// TIA Portal V17 program export: 0 tag tables, 0 data types, 15 data blocks, 22 code blocks (in call order from the OBs), 17 instance data blocks

DATA_BLOCK "GLOBAL_DB"   // DB14
{ S7_Optimized_Access := 'TRUE' }
VERSION : 0.1
// stored: AutoNumber true, DBAccessibleFromOPCUA true, DBAccessibleFromWebserver true, IsOnlyStoredInLoadMemory false, IsRetainMemResEnabled false, IsWriteProtectedInAS false, MemoryReserve 100
   VAR
      CurrentTime : Date_And_Time;
      RS232_SendBuff : DWord;
      RS232_RecvBuff : DWord;
   END_VAR
BEGIN
END_DATA_BLOCK

DATA_BLOCK "GDB_Database"   // DB7
{ S7_Optimized_Access := 'TRUE' }
VERSION : 0.1
// stored: AutoNumber true, DBAccessibleFromOPCUA true, DBAccessibleFromWebserver true, IsOnlyStoredInLoadMemory false, IsRetainMemResEnabled false, IsWriteProtectedInAS false, MemoryReserve 100
   VAR
      Communication : Struct   // Communication_Status
         Error : Int;
         Active : Bool;
         Start : Bool;
         Function : Int;
         "Step" : Int;
         Done : Int;
      END_STRUCT;
      Condition : Struct
         Rob_PrgNmr : Int;
      END_STRUCT;
      Receive : Struct
         Rob_PRG : Int;
         Force : Real;
      END_STRUCT;
      Task_Done : Struct
         Read_from_DB : Bool;
      END_STRUCT;
      "Return" : Struct
         t : Bool;
      END_STRUCT;
      Requests : Struct
         Read_from_DB : Bool;
         Write_to_DB : Bool;
      END_STRUCT;
   END_VAR
BEGIN
END_DATA_BLOCK

DATA_BLOCK "STL_Data"   // DB2
{ S7_Optimized_Access := 'TRUE' }
VERSION : 0.1
// stored: AutoNumber true, DBAccessibleFromOPCUA true, DBAccessibleFromWebserver true, IsOnlyStoredInLoadMemory false, IsRetainMemResEnabled false, IsWriteProtectedInAS false, MemoryReserve 100
   VAR
      BasePos0 : Int;
      BasePos1 : Int;
      VarBase0 : Int;
      VarBase1 : Int;
   END_VAR
BEGIN
END_DATA_BLOCK

DATA_BLOCK "DATA_LOGGING"   // DB25
{ S7_Optimized_Access := 'TRUE' }
VERSION : 0.1
// stored: AutoNumber true, DBAccessibleFromOPCUA true, DBAccessibleFromWebserver true, IsOnlyStoredInLoadMemory false, IsRetainMemResEnabled false, IsWriteProtectedInAS false, MemoryReserve 100
   VAR
      Record : UDInt;
      "Name" : String := 'Logging';
      ID : DWord := 1;
      Header : String := 'A350-1000, Errors';
      Data : Struct
         First : UDInt;
         Second : UDInt;
         Third : UDInt;
      END_STRUCT;
   END_VAR
BEGIN
END_DATA_BLOCK

DATA_BLOCK "GDB_HMI"   // DB8
{ S7_Optimized_Access := 'TRUE' }
VERSION : 0.1
// stored: AutoNumber true, DBAccessibleFromOPCUA true, DBAccessibleFromWebserver true, IsOnlyStoredInLoadMemory false, IsRetainMemResEnabled false, IsWriteProtectedInAS false, MemoryReserve 100
   VAR
      Database : Struct
         Reset_Task : Bool;
      END_STRUCT;
      Received_Data_from_DB : Struct
         Rob_PRG : Int;
         Force : Real;
      END_STRUCT;
   END_VAR
BEGIN
END_DATA_BLOCK

DATA_BLOCK "ProjectDB78"   // DB30
{ S7_Optimized_Access := 'FALSE' }
VERSION : 0.1
// stored: AutoNumber true, DBAccessibleFromOPCUA true, DBAccessibleFromWebserver true, IsOnlyStoredInLoadMemory false, IsWriteProtectedInAS false
   VAR
      Oven_Temperature : Array[1..2100] of "OvenTemperature";
   END_VAR
BEGIN
END_DATA_BLOCK

DATA_BLOCK "ProjectDB94"   // DB29
{ S7_Optimized_Access := 'FALSE' }
VERSION : 0.1
// stored: AutoNumber true, DBAccessibleFromOPCUA true, DBAccessibleFromWebserver true, IsOnlyStoredInLoadMemory false, IsWriteProtectedInAS false
   VAR
      MainDB : "OvenTemperature";
      Req_Start { S7_SetPoint := 'True'} : Bool;
      Archive_Done : Bool;
   END_VAR
BEGIN
END_DATA_BLOCK

DATA_BLOCK "Keyence Datenausgabe"   // DB4
{ S7_Optimized_Access := 'TRUE' }
VERSION : 0.1
// stored: AutoNumber true, DBAccessibleFromOPCUA true, DBAccessibleFromWebserver true, IsOnlyStoredInLoadMemory false, IsRetainMemResEnabled false, IsWriteProtectedInAS false, MemoryReserve 100
   VAR
      Breite : Int;
      Länge : Int;
      Länge1 : Real;
      Breite1 : Real;
   END_VAR
BEGIN
END_DATA_BLOCK

DATA_BLOCK "DB_CMMT_ST"   // DB13
{ S7_Optimized_Access := 'TRUE' }
VERSION : 0.1
// stored: AutoNumber true, DBAccessibleFromOPCUA true, DBAccessibleFromWebserver true, IsOnlyStoredInLoadMemory false, IsRetainMemResEnabled false, IsWriteProtectedInAS false, MemoryReserve 100
   VAR
      "PLC -> CMMT" : "UDT_FESTO_CMMT_IN";
      "CMMT -> PLC" { S7_SetPoint := 'True'} : "UDT_FESTO_CMMT_OUT";
      ActualPos_mm { S7_SetPoint := 'True'} : Real;
      AcutalVelocity_mm_s : Real;
      SetPosition_mm : Real;
      SetVelocity_mm_s : Real := 20.0;
      HMI : Struct
         Scaled_ActualPos : Real;
         Scaled_SetpointPosition : Real;
         Scaled_ActualVelocity : Real;
      END_STRUCT;
      CLAMPING_TORQUE : Struct
         Execute : Bool;
         LinearRotative : Bool;
         ClampingTorque : Real;
         PercentForce : Real;
      END_STRUCT;
      CMMT_ST_ErrorWarningMessage : String;
   END_VAR
BEGIN
   "PLC -> CMMT".CancelTraversing := TRUE;
   "PLC -> CMMT".IntermediateStop := TRUE;
   "PLC -> CMMT".OverV := 100;
   "PLC -> CMMT".BaseSpeedValue := 0.125;
END_DATA_BLOCK

DATA_BLOCK "GDB_LJ_X8000"   // DB10
{ S7_Optimized_Access := 'TRUE' }
VERSION : 0.1
// stored: AutoNumber true, DBAccessibleFromOPCUA true, DBAccessibleFromWebserver true, IsOnlyStoredInLoadMemory false, IsRetainMemResEnabled false, IsWriteProtectedInAS false, MemoryReserve 100
   VAR
      PLC_to_LJX8000bits : "UDT_PLC --> LJ_X8000_Bits";
      PLC_to_LJX8000bytes { S7_SetPoint := 'True'} : "UDT_PLC --> LJ_X8000_Bytes";
      LJX8000_to_PLCbits { S7_SetPoint := 'True'} : "UDT_LJ_X8000 --> PLC_Bits";
      LJX8000_to_PLCbytes { S7_SetPoint := 'True'} : "UDT_LJ_X8000 --> PLC_Bytes";
      CTRL : Struct
         UserCommand : Int;
         ProgramNumber : Int;
         ResetError : Bool;
         CommandRequest : Bool;
         Trigger : Bool;
      END_STRUCT;
      HMI : Struct
         StartMeasurement : Bool;
         MeasurementMode : Bool;
         HandMode : Bool;
         CellType : SInt;
         SQ_ActivTask : SInt;
      END_STRUCT;
      Cell_MeasData : Struct
         Länge : Real;
         Breite : Real;
      END_STRUCT;
   END_VAR
BEGIN
END_DATA_BLOCK

DATA_BLOCK "Global_Data"   // DB3
{ S7_Optimized_Access := 'TRUE' }
VERSION : 0.1
// stored: AutoNumber true, DBAccessibleFromOPCUA true, DBAccessibleFromWebserver true, IsOnlyStoredInLoadMemory false, IsRetainMemResEnabled false, IsWriteProtectedInAS false, MemoryReserve 100
   VAR
      "LK-G5001P" : Struct   // Distanzsensoren - KEYENCE
         "LK-H057-01" : Real;
         "LK-H057-02" : Real;
      END_STRUCT;
      testbit : Bool;
   END_VAR
BEGIN
END_DATA_BLOCK

DATA_BLOCK "LK_G5000_DATA"   // DB16
{ S7_Optimized_Access := 'TRUE' }
VERSION : 0.1
// stored: AutoNumber true, DBAccessibleFromOPCUA true, DBAccessibleFromWebserver true, IsOnlyStoredInLoadMemory false, IsRetainMemResEnabled false, IsWriteProtectedInAS false, MemoryReserve 100
   VAR
      RS232_CTRL : Struct
         TO_LKG5000 : "UDT_LKG5000_RS232_SEND";
         FROM_LKG5000 { S7_SetPoint := 'True'} : "UDT_LKG5000_RS232_RCV";
      END_STRUCT;
      SEND_BUFF : "UDT_RS232_SEND_DATA";
      RCV_BUFF { S7_SetPoint := 'True'} : "UDT_RS232_RCV_DATA";
      RS232_Command { S7_SetPoint := 'True'} : String[11];
   END_VAR
BEGIN
END_DATA_BLOCK

DATA_BLOCK "DB_Receipe"   // DB6
{ S7_Optimized_Access := 'TRUE' }
VERSION : 0.1
// stored: AutoNumber true, DBAccessibleFromOPCUA true, DBAccessibleFromWebserver true, IsOnlyStoredInLoadMemory false, IsRetainMemResEnabled false, IsWriteProtectedInAS false, MemoryReserve 100
   VAR
      "Time" : Time;
      Temperature : Int;
      Fan : Bool;
   END_VAR
BEGIN
END_DATA_BLOCK

DATA_BLOCK "DB_ScanData"   // DB5
{ S7_Optimized_Access := 'TRUE' }
VERSION : 0.1
// stored: AutoNumber true, DBAccessibleFromOPCUA true, DBAccessibleFromWebserver true, IsOnlyStoredInLoadMemory false, IsRetainMemResEnabled false, IsWriteProtectedInAS false, MemoryReserve 100
   VAR
      ST01_MessGewichtMasse : Struct
         Request_for_Scan : Bool;
         DatenVorhanden : Bool;
         "Tray+Zelle" : Array[1..1, 1..1] of "UDT_ProGloveScanDat";
      END_STRUCT;
      ST02_EOLMessungImpdanz : Struct
         Request_for_Scan : Bool;
         DatenVoranden : Bool;
         "Tray+Zelle" : Array[1..2, 1..6] of "UDT_ProGloveScanDat";
      END_STRUCT;
      ST03_Dichtigkeitspruefung : Struct
         Request_for_Scan : Bool;
         DatenVoranden : Bool;
         "Tray+Zelle" : Array[1..1, 1..1] of "UDT_ProGloveScanDat";
      END_STRUCT;
      ST04_Degassing : Struct
         Request_for_Scan : Bool;
         DatenVorhanden : Bool;
         "Tray+Zelle" : Array[1..1, 1..1] of "UDT_ProGloveScanDat";
      END_STRUCT;
      ST05_Formierung : Struct
         Request_for_Scan : Bool;
         DatenVorhanden : Bool;
         Schrank : Array[1..2] of "UDT_Formierung";
      END_STRUCT;
      ST06_Soaking : Struct
         Request_for_Scan : Bool;
         DatenVorhanden : Bool;
         Schrank : Array[1..4] of "UDT_Formierung";
      END_STRUCT;
      ST07_Aging : Struct
         Request_for_Scan : Bool;
         DatenVorhanden : Bool;
         Schrank : Array[1..30] of "UDT_Aging";
      END_STRUCT;
      ST08_MobileOCVMessung : Struct
         Request_for_Scan : Bool;
         DatenVorhanden : Bool;
         "Tray+Zelle" : Array[1..1, 1..6] of "UDT_ProGloveScanDat";
      END_STRUCT;
   END_VAR
BEGIN
END_DATA_BLOCK

DATA_BLOCK "PROGLOVE_TCP"   // DB32
{ S7_Optimized_Access := 'TRUE' }
VERSION : 0.1
// stored: AutoNumber true, DBAccessibleFromOPCUA true, DBAccessibleFromWebserver true, IsOnlyStoredInLoadMemory false, IsRetainMemResEnabled false, IsWriteProtectedInAS false, MemoryReserve 100
   VAR
      SEND_DATA { S7_SetPoint := 'True'} : String;
      RCV_DATA : String;
      TCON : Struct
         Done : Bool;
         Busy : Bool;
         Error : Bool;
         Status : Word;
      END_STRUCT;
   END_VAR
BEGIN
END_DATA_BLOCK

ORGANIZATION_BLOCK "Main"   // OB1, LAD, ProgramCycle
TITLE = "Main Program Sweep (Cycle)"
{ S7_Optimized_Access := 'TRUE' }
VERSION : 0.1
// stored: AutoNumber true, IsIECCheckEnabled false, SetENOAutomatically false
   VAR_INPUT
      Initial_Call : Bool;   // Initial call of this OB
      Remanence : Bool;   // =True, if remanent data are available
   END_VAR
   VAR_TEMP
      RetVAl : Int;
   END_VAR
BEGIN

REGION Network 1: Read Local Time
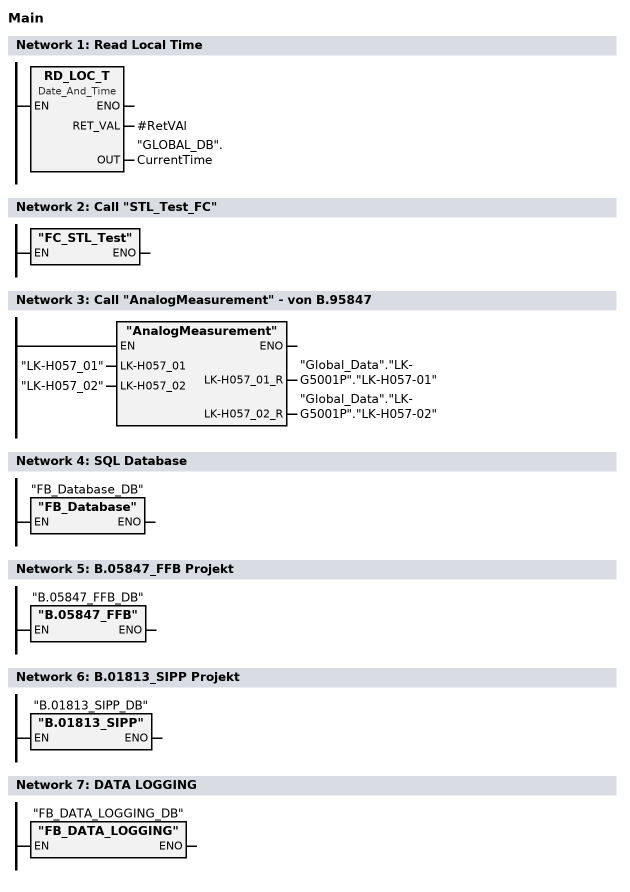
   RUNG wire#powerrail
      { S7_Templates := "date_type := Date_And_Time" } RD_LOC_T(RET_VAL => #RetVAl, OUT => "GLOBAL_DB".CurrentTime)
   END_RUNG
   // the same network as SCL:
   #RetVAl := RD_LOC_T(OUT => "GLOBAL_DB".CurrentTime);
END_REGION

REGION Network 2: Call "STL_Test_FC"
   RUNG wire#powerrail
      "FC_STL_Test"()
   END_RUNG
   // the same network as SCL:
   "FC_STL_Test"();
END_REGION

REGION Network 3: Call "AnalogMeasurement" - von B.95847
   RUNG wire#powerrail
      "AnalogMeasurement"("LK-H057_01" := "LK-H057_01", "LK-H057_02" := "LK-H057_02", "LK-H057_01_R" => "Global_Data"."LK-G5001P"."LK-H057-01", "LK-H057_02_R" => "Global_Data"."LK-G5001P"."LK-H057-02")
   END_RUNG
   // the same network as SCL:
   "AnalogMeasurement"("LK-H057_01" := "LK-H057_01",
                       "LK-H057_02" := "LK-H057_02",
                       "LK-H057_01_R" => "Global_Data"."LK-G5001P"."LK-H057-01",
                       "LK-H057_02_R" => "Global_Data"."LK-G5001P"."LK-H057-02");
END_REGION

REGION Network 4: SQL Database
   RUNG wire#powerrail
      "FB_Database_DB"()
   END_RUNG
   // the same network as SCL:
   "FB_Database_DB"();   // "FB_Database"
END_REGION

REGION Network 5: B.05847_FFB Projekt
   RUNG wire#powerrail
      "B.05847_FFB_DB"()
   END_RUNG
   // the same network as SCL:
   "B.05847_FFB_DB"();   // "B.05847_FFB"
END_REGION

REGION Network 6: B.01813_SIPP Projekt
   RUNG wire#powerrail
      "B.01813_SIPP_DB"()
   END_RUNG
   // the same network as SCL:
   "B.01813_SIPP_DB"();   // "B.01813_SIPP"
END_REGION

REGION Network 7: DATA LOGGING
   RUNG wire#powerrail
      "FB_DATA_LOGGING_DB"()
   END_RUNG
   // the same network as SCL:
   "FB_DATA_LOGGING_DB"();   // "FB_DATA_LOGGING"
END_REGION
END_ORGANIZATION_BLOCK

FUNCTION "FC_STL_Test" : Void   // FC1, STL
{ S7_Optimized_Access := 'TRUE' }
VERSION : 0.1
// stored: AutoNumber true, UDAEnableTagReadback false
BEGIN

NETWORK
TITLE = 
// Example how to Load Set values to ACC1 ( defined variable by T )
// L is for LOAD
// T is for TRANSFER the value from bottom ( L )

      L     125;
      T     "STL_Data".BasePos0;

      L     "STL_Data".VarBase1;
      T     "STL_Data".BasePos1;


END_FUNCTION

FUNCTION "AnalogMeasurement" : Void   // FC2, LAD
{ S7_Optimized_Access := 'TRUE' }
VERSION : 0.1
// stored: AutoNumber true, IsIECCheckEnabled false, SetENOAutomatically false, UDAEnableTagReadback false
   VAR_INPUT
      "LK-H057_01" : Int;   // Keyence Dist.Senz-01
      "LK-H057_02" : Int;   // Keyence Dist.Senz-01
   END_VAR
   VAR_OUTPUT
      "LK-H057_01_R" : Real;
      "LK-H057_02_R" : Real;
   END_VAR
   VAR_TEMP
      Distanz_In_Prozent_01 : Real;
      Distanz_In_Prozent_02 : Real;
   END_VAR
BEGIN

REGION Network 1: LK-H057_01 Analog Werte
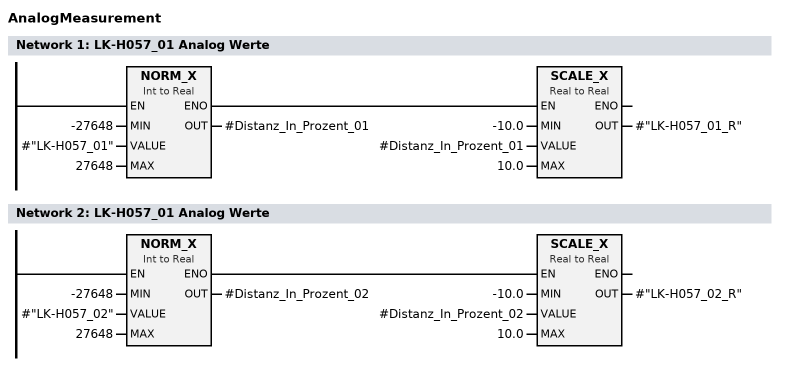
   RUNG wire#powerrail
      { S7_Templates := "[SrcType := Int, DestType := Real]" } Normalize(min := -27648, value := #"LK-H057_01", max := 27648, out => #Distanz_In_Prozent_01)
      { S7_Templates := "[SrcType := Real, DestType := Real]" } Scale(min := -10.0, value := #Distanz_In_Prozent_01, max := 10.0, out => #"LK-H057_01_R")
   END_RUNG
   // the same network as SCL:
   #Distanz_In_Prozent_01 := NORM_X(MIN := -27648, VALUE := #"LK-H057_01", MAX := 27648);
   #"LK-H057_01_R" := SCALE_X(MIN := -10.0, VALUE := #Distanz_In_Prozent_01, MAX := 10.0);
END_REGION

REGION Network 2: LK-H057_01 Analog Werte
   RUNG wire#powerrail
      { S7_Templates := "[SrcType := Int, DestType := Real]" } Normalize(min := -27648, value := #"LK-H057_02", max := 27648, out => #Distanz_In_Prozent_02)
      { S7_Templates := "[SrcType := Real, DestType := Real]" } Scale(min := -10.0, value := #Distanz_In_Prozent_02, max := 10.0, out => #"LK-H057_02_R")
   END_RUNG
   // the same network as SCL:
   #Distanz_In_Prozent_02 := NORM_X(MIN := -27648, VALUE := #"LK-H057_02", MAX := 27648);
   #"LK-H057_02_R" := SCALE_X(MIN := -10.0, VALUE := #Distanz_In_Prozent_02, MAX := 10.0);
END_REGION
END_FUNCTION

FUNCTION_BLOCK "FB_Database"   // FB2, LAD
{ S7_Optimized_Access := 'TRUE' }
VERSION : 0.1
// stored: AutoNumber true, IsIECCheckEnabled false, IsRetainMemResEnabled false, MemoryReserve 100, SetENOAutomatically false, UDAEnableTagReadback false
   VAR
      task : Int;
      Task_Start : Bool;
      TON_Act_Script { S7_SetPoint := 'True'} : TON_TIME;
   END_VAR
   VAR_TEMP
      Request : Struct
         Task_001 : Bool;
         Task_002 : Bool;
         Task_003 : Bool;
         Task_004 : Bool;
      END_STRUCT;
   END_VAR
   VAR CONSTANT
      S001_Get_Data : Int := 1;
      S002_Write_Data : Int := 2;
   END_VAR
BEGIN

NETWORK
TITLE = Reset Task Requests
// Reset Task Requests
      A     "GDB_HMI".Database.Reset_Task;
      R     "GDB_Database".Requests.Read_from_DB;
      R     "GDB_Database".Requests.Write_to_DB;



REGION Network 2 (SCL): Task Start Request
   #Request.Task_001 := "GDB_Database".Requests.Read_from_DB;
   #Request.Task_002 := "GDB_Database".Requests.Write_to_DB;
END_REGION

REGION Network 3 (SCL): 10 = Request for read Global Data
   // Set task
   IF #Request.Task_001 AND (#task = 0) THEN
       #task := 10;
   END_IF;


   //Fullfill task
   IF #task = 10 THEN

       // If reading is done
       IF "GDB_Database".Communication.Done = #S001_Get_Data AND NOT "GDB_Database".Task_Done.Read_from_DB AND "GDB_Database".Communication.Error = 0 THEN

           // Write Data from DB Receive ( on HMI Tags ) to DB on SPS
          // "GDB_HMI".Received_Data_from_DB.Rob_PRG := "GDB_Database".Receive.Rob_PRG;
          // "GDB_HMI".Received_Data_from_DB.Force := "GDB_Database".Receive.Force;
           // Set that Task is active
           "GDB_Database".Task_Done.Read_from_DB := TRUE;

       END_IF;

       // Control script
       IF #Request.Task_001 THEN
           "GDB_Database".Communication.Function := #S001_Get_Data;
           #Task_Start := TRUE;
       ELSE
           "GDB_Database".Communication.Function := 0;
           #Task_Start := FALSE;
           IF NOT "GDB_Database".Communication.Active AND "GDB_Database".Communication.Done = 0 THEN
               #task := 0;
           END_IF;
       END_IF;
   END_IF;

   // Reset Done
   IF NOT #Request.Task_001 THEN
       "GDB_Database".Task_Done.Read_from_DB := FALSE;
   END_IF;
END_REGION

REGION Network 4
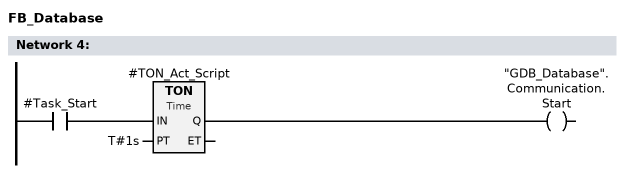
   RUNG wire#powerrail
      Contact( #Task_Start )
      { S7_Templates := "time_type := Time" } #TON_Act_Script.TON(pt := T#1s, et =>)
      Coil( "GDB_Database".Communication.Start )
   END_RUNG
   // the same network as SCL:
   #TON_Act_Script(IN := #Task_Start, PT := T#1s);   // TON
   "GDB_Database".Communication.Start := #TON_Act_Script.Q;
END_REGION
END_FUNCTION_BLOCK

FUNCTION_BLOCK "B.05847_FFB"   // FB3, LAD
{ S7_Optimized_Access := 'TRUE' }
VERSION : 0.1
// stored: AutoNumber true, IsIECCheckEnabled false, IsRetainMemResEnabled false, MemoryReserve 100, SetENOAutomatically false, UDAEnableTagReadback false
BEGIN

REGION Network 1: FESTO_CMMT_ST
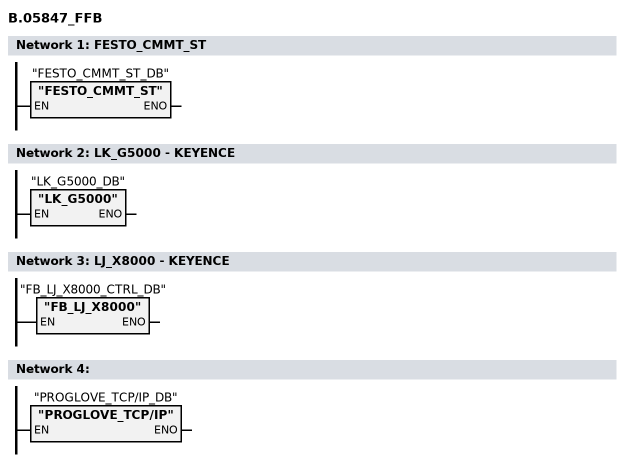
   RUNG wire#powerrail
      "FESTO_CMMT_ST_DB"()
   END_RUNG
   // the same network as SCL:
   "FESTO_CMMT_ST_DB"();   // "FESTO_CMMT_ST"
END_REGION

REGION Network 2: LK_G5000 - KEYENCE
   RUNG wire#powerrail
      "LK_G5000_DB"()
   END_RUNG
   // the same network as SCL:
   "LK_G5000_DB"();   // "LK_G5000"
END_REGION

REGION Network 3: LJ_X8000 - KEYENCE
   RUNG wire#powerrail
      "FB_LJ_X8000_CTRL_DB"()
   END_RUNG
   // the same network as SCL:
   "FB_LJ_X8000_CTRL_DB"();   // "FB_LJ_X8000"
END_REGION

REGION Network 4
   RUNG wire#powerrail
      "PROGLOVE_TCP/IP_DB"()
   END_RUNG
   // the same network as SCL:
   "PROGLOVE_TCP/IP_DB"();   // "PROGLOVE_TCP/IP"
END_REGION
END_FUNCTION_BLOCK

FUNCTION_BLOCK "FESTO_CMMT_ST"   // FB4, LAD
{ S7_Optimized_Access := 'TRUE' }
VERSION : 0.1
// stored: AutoNumber true, IsIECCheckEnabled false, IsRetainMemResEnabled false, MemoryReserve 100, SetENOAutomatically false, UDAEnableTagReadback false
   VAR
      Festo_PtP_Drives_PN_Instance { S7_SetPoint := 'True'} : "Festo_PtP_Drives_PN";
   END_VAR
   VAR_TEMP
      i : Int;
   END_VAR
BEGIN

REGION Network 1
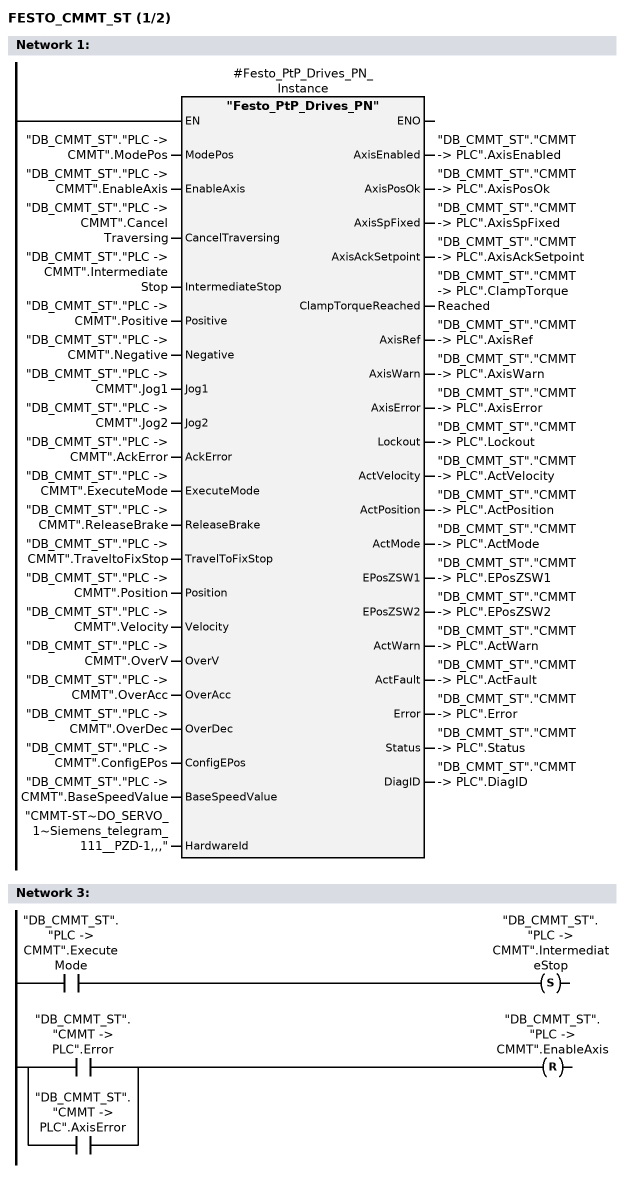
   RUNG wire#powerrail
      #Festo_PtP_Drives_PN_Instance(ModePos := "DB_CMMT_ST"."PLC -> CMMT".ModePos, EnableAxis := "DB_CMMT_ST"."PLC -> CMMT".EnableAxis, CancelTraversing := "DB_CMMT_ST"."PLC -> CMMT".CancelTraversing, IntermediateStop := "DB_CMMT_ST"."PLC -> CMMT".IntermediateStop, Positive := "DB_CMMT_ST"."PLC -> CMMT".Positive, Negative := "DB_CMMT_ST"."PLC -> CMMT".Negative, Jog1 := "DB_CMMT_ST"."PLC -> CMMT".Jog1, Jog2 := "DB_CMMT_ST"."PLC -> CMMT".Jog2, AckError := "DB_CMMT_ST"."PLC -> CMMT".AckError, ExecuteMode := "DB_CMMT_ST"."PLC -> CMMT".ExecuteMode, ReleaseBrake := "DB_CMMT_ST"."PLC -> CMMT".ReleaseBrake, TravelToFixStop := "DB_CMMT_ST"."PLC -> CMMT".TraveltoFixStop, Position := "DB_CMMT_ST"."PLC -> CMMT".Position, Velocity := "DB_CMMT_ST"."PLC -> CMMT".Velocity, OverV := "DB_CMMT_ST"."PLC -> CMMT".OverV, OverAcc := "DB_CMMT_ST"."PLC -> CMMT".OverAcc, OverDec := "DB_CMMT_ST"."PLC -> CMMT".OverDec, ConfigEPos := "DB_CMMT_ST"."PLC -> CMMT".ConfigEPos, BaseSpeedValue := "DB_CMMT_ST"."PLC -> CMMT".BaseSpeedValue, HardwareId := "CMMT-ST~DO_SERVO_1~Siemens_telegram_111__PZD-1,,,", AxisEnabled => "DB_CMMT_ST"."CMMT -> PLC".AxisEnabled, AxisPosOk => "DB_CMMT_ST"."CMMT -> PLC".AxisPosOk, AxisSpFixed => "DB_CMMT_ST"."CMMT -> PLC".AxisSpFixed, AxisAckSetpoint => "DB_CMMT_ST"."CMMT -> PLC".AxisAckSetpoint, ClampTorqueReached => "DB_CMMT_ST"."CMMT -> PLC".ClampTorqueReached, AxisRef => "DB_CMMT_ST"."CMMT -> PLC".AxisRef, AxisWarn => "DB_CMMT_ST"."CMMT -> PLC".AxisWarn, AxisError => "DB_CMMT_ST"."CMMT -> PLC".AxisError, Lockout => "DB_CMMT_ST"."CMMT -> PLC".Lockout, ActVelocity => "DB_CMMT_ST"."CMMT -> PLC".ActVelocity, ActPosition => "DB_CMMT_ST"."CMMT -> PLC".ActPosition, ActMode => "DB_CMMT_ST"."CMMT -> PLC".ActMode, EPosZSW1 => "DB_CMMT_ST"."CMMT -> PLC".EPosZSW1, EPosZSW2 => "DB_CMMT_ST"."CMMT -> PLC".EPosZSW2, ActWarn => "DB_CMMT_ST"."CMMT -> PLC".ActWarn, ActFault => "DB_CMMT_ST"."CMMT -> PLC".ActFault, Error => "DB_CMMT_ST"."CMMT -> PLC".Error, Status => "DB_CMMT_ST"."CMMT -> PLC".Status, DiagID => "DB_CMMT_ST"."CMMT -> PLC".DiagID)
   END_RUNG
   // the same network as SCL:
   #Festo_PtP_Drives_PN_Instance(ModePos := "DB_CMMT_ST"."PLC -> CMMT".ModePos,   // "Festo_PtP_Drives_PN"
                           EnableAxis := "DB_CMMT_ST"."PLC -> CMMT".EnableAxis,
                           CancelTraversing := "DB_CMMT_ST"."PLC -> CMMT".CancelTraversing,
                           IntermediateStop := "DB_CMMT_ST"."PLC -> CMMT".IntermediateStop,
                           Positive := "DB_CMMT_ST"."PLC -> CMMT".Positive,
                           Negative := "DB_CMMT_ST"."PLC -> CMMT".Negative,
                           Jog1 := "DB_CMMT_ST"."PLC -> CMMT".Jog1,
                           Jog2 := "DB_CMMT_ST"."PLC -> CMMT".Jog2,
                           AckError := "DB_CMMT_ST"."PLC -> CMMT".AckError,
                           ExecuteMode := "DB_CMMT_ST"."PLC -> CMMT".ExecuteMode,
                           ReleaseBrake := "DB_CMMT_ST"."PLC -> CMMT".ReleaseBrake,
                           TravelToFixStop := "DB_CMMT_ST"."PLC -> CMMT".TraveltoFixStop,
                           Position := "DB_CMMT_ST"."PLC -> CMMT".Position,
                           Velocity := "DB_CMMT_ST"."PLC -> CMMT".Velocity,
                           OverV := "DB_CMMT_ST"."PLC -> CMMT".OverV,
                           OverAcc := "DB_CMMT_ST"."PLC -> CMMT".OverAcc,
                           OverDec := "DB_CMMT_ST"."PLC -> CMMT".OverDec,
                           ConfigEPos := "DB_CMMT_ST"."PLC -> CMMT".ConfigEPos,
                           BaseSpeedValue := "DB_CMMT_ST"."PLC -> CMMT".BaseSpeedValue,
                           HardwareId := "CMMT-ST~DO_SERVO_1~Siemens_telegram_111__PZD-1,,,",
                           AxisEnabled => "DB_CMMT_ST"."CMMT -> PLC".AxisEnabled,
                           AxisPosOk => "DB_CMMT_ST"."CMMT -> PLC".AxisPosOk,
                           AxisSpFixed => "DB_CMMT_ST"."CMMT -> PLC".AxisSpFixed,
                           AxisAckSetpoint => "DB_CMMT_ST"."CMMT -> PLC".AxisAckSetpoint,
                           ClampTorqueReached => "DB_CMMT_ST"."CMMT -> PLC".ClampTorqueReached,
                           AxisRef => "DB_CMMT_ST"."CMMT -> PLC".AxisRef,
                           AxisWarn => "DB_CMMT_ST"."CMMT -> PLC".AxisWarn,
                           AxisError => "DB_CMMT_ST"."CMMT -> PLC".AxisError,
                           Lockout => "DB_CMMT_ST"."CMMT -> PLC".Lockout,
                           ActVelocity => "DB_CMMT_ST"."CMMT -> PLC".ActVelocity,
                           ActPosition => "DB_CMMT_ST"."CMMT -> PLC".ActPosition,
                           ActMode => "DB_CMMT_ST"."CMMT -> PLC".ActMode,
                           EPosZSW1 => "DB_CMMT_ST"."CMMT -> PLC".EPosZSW1,
                           EPosZSW2 => "DB_CMMT_ST"."CMMT -> PLC".EPosZSW2,
                           ActWarn => "DB_CMMT_ST"."CMMT -> PLC".ActWarn,
                           ActFault => "DB_CMMT_ST"."CMMT -> PLC".ActFault,
                           Error => "DB_CMMT_ST"."CMMT -> PLC".Error,
                           Status => "DB_CMMT_ST"."CMMT -> PLC".Status,
                           DiagID => "DB_CMMT_ST"."CMMT -> PLC".DiagID);
END_REGION

REGION Network 2 (SCL): Convert Veolocity and Position in mm/s and mm
   REGION Convert Setposition from mm TO 1000_Unit
       "DB_CMMT_ST"."PLC -> CMMT".Position   := REAL_TO_DINT("DB_CMMT_ST".SetPosition_mm * 1000.0);
       "DB_CMMT_ST".HMI.Scaled_SetpointPosition := "DB_CMMT_ST".SetPosition_mm / 100.0;
   END_REGION

   REGION Convert Setvelocity 
       "DB_CMMT_ST"."PLC -> CMMT".Velocity := REAL_TO_DINT("DB_CMMT_ST".SetVelocity_mm_s);
   END_REGION

   REGION Convert Actual Position from 1000Unit to mm
       "DB_CMMT_ST".ActualPos_mm := "DB_CMMT_ST"."CMMT -> PLC".ActPosition / 1000.0;
       // Scale actual position for HMI
       "DB_CMMT_ST".HMI.Scaled_ActualPos := "DB_CMMT_ST".ActualPos_mm / 100; // Value in cm
   END_REGION

   REGION Convert Actual velocity from 1000Unit TO mm/s
       "DB_CMMT_ST".AcutalVelocity_mm_s := "DB_CMMT_ST"."CMMT -> PLC".ActVelocity * 1000.0;
   END_REGION
END_REGION

REGION Network 3
   RUNG wire#powerrail
      Contact( "DB_CMMT_ST"."PLC -> CMMT".ExecuteMode )
      S_Coil( "DB_CMMT_ST"."PLC -> CMMT".IntermediateStop )
   END_RUNG
   RUNG wire#powerrail
      Contact( "DB_CMMT_ST"."CMMT -> PLC".Error )
      wire#w1
      R_Coil( "DB_CMMT_ST"."PLC -> CMMT".EnableAxis )
   END_RUNG
   RUNG wire#powerrail
      Contact( "DB_CMMT_ST"."CMMT -> PLC".AxisError )
   END_RUNG wire#w1
   // the same network as SCL:
   IF "DB_CMMT_ST"."PLC -> CMMT".ExecuteMode THEN
       "DB_CMMT_ST"."PLC -> CMMT".IntermediateStop := TRUE;
   END_IF;
   IF "DB_CMMT_ST"."CMMT -> PLC".Error OR "DB_CMMT_ST"."CMMT -> PLC".AxisError THEN
       "DB_CMMT_ST"."PLC -> CMMT".EnableAxis := FALSE;
   END_IF;
END_REGION

REGION Network 4: Festo Calmping Torque
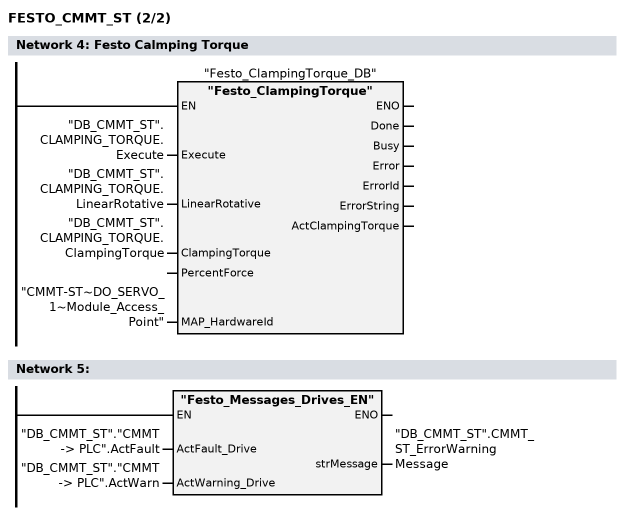
   RUNG wire#powerrail
      "Festo_ClampingTorque_DB"(Execute := "DB_CMMT_ST".CLAMPING_TORQUE.Execute, LinearRotative := "DB_CMMT_ST".CLAMPING_TORQUE.LinearRotative, ClampingTorque := "DB_CMMT_ST".CLAMPING_TORQUE.ClampingTorque, PercentForce :=, MAP_HardwareId := "CMMT-ST~DO_SERVO_1~Module_Access_Point", Done =>, Busy =>, Error =>, ErrorId =>, ErrorString =>, ActClampingTorque =>)
   END_RUNG
   // the same network as SCL:
   "Festo_ClampingTorque_DB"(Execute := "DB_CMMT_ST".CLAMPING_TORQUE.Execute,   // "Festo_ClampingTorque"
                           LinearRotative := "DB_CMMT_ST".CLAMPING_TORQUE.LinearRotative,
                           ClampingTorque := "DB_CMMT_ST".CLAMPING_TORQUE.ClampingTorque,
                           MAP_HardwareId := "CMMT-ST~DO_SERVO_1~Module_Access_Point");
END_REGION

REGION Network 5
   RUNG wire#powerrail
      "Festo_Messages_Drives_EN"(ActFault_Drive := "DB_CMMT_ST"."CMMT -> PLC".ActFault, ActWarning_Drive := "DB_CMMT_ST"."CMMT -> PLC".ActWarn, strMessage => "DB_CMMT_ST".CMMT_ST_ErrorWarningMessage)
   END_RUNG
   // the same network as SCL:
   "Festo_Messages_Drives_EN"(ActFault_Drive := "DB_CMMT_ST"."CMMT -> PLC".ActFault,
                           ActWarning_Drive := "DB_CMMT_ST"."CMMT -> PLC".ActWarn,
                           strMessage => "DB_CMMT_ST".CMMT_ST_ErrorWarningMessage);
END_REGION
END_FUNCTION_BLOCK

FUNCTION_BLOCK "Festo_PtP_Drives_PN"
TITLE = PtP function block for positioning with Tel111
{ S7_Optimized_Access := 'TRUE' }
AUTHOR : Festo
FAMILY : 'E-.Drives'
VERSION : 1.5
   VAR_INPUT 
      ModePos : Int := 0;   //   Settings of the mode
      EnableAxis : Bool := 0;   //   1 = Enable the drive
      CancelTraversing : Bool := 1;   //   0 = Reject active traverse task
      IntermediateStop : Bool := 1;   //   0 = IntermediateStop
      Positive : Bool := 0;   //   1 = Modulo positive
      Negative : Bool := 0;   //   1 = Modulo negative
      Jog1 : Bool := 0;   //   1 = jog positive
      Jog2 : Bool := 0;   //   1 = jog negative
      AckError : Bool := 0;   //   1  = Acknowledge of errors
      ExecuteMode : Bool := 0;   //   0-->1 = Start the mode
      ReleaseBrake : Bool := 0;   //   1 = Release Brake 0 = close
      TravelToFixStop : Bool := 0;   //   1 = Activation TravelToFixStop
      Position : DInt := 0;   //   Position of the MDI mode or setting of traversing block
      Velocity : DInt := 0;   //   MDI velocity
      OverV : Int := 100;   //   Override of  velocity in [%] --> 4000h=100%
      OverAcc : Int := 100;   //   Override of acceleration in [%] --> 4000h=100%
      OverDec : Int := 100;   //   Override of deceleration in [%] --> 4000h=100%
      ConfigEPos : DWord := 16#0000_000F;   //   binary programmed input -> see manual
      BaseSpeedValue : Real;   //   Value for scaling the RPM display value
      HardwareId : HW_IO := 0;   //   Hardware Identifer
   END_VAR

   VAR_OUTPUT 
      AxisEnabled : Bool := 0;   //   1= Axis in operation
      AxisPosOk : Bool := 0;   //   1= Position setpoint reached
      AxisSpFixed : Bool := 0;   //   1= Drive at standstill
      AxisAckSetpoint : Bool := 0;   //   1= Acknowledge setpoint
      ClampTorqueReached : Bool;   //   1= Clamping torque is reached
      AxisRef : Bool := 0;   //   1= Reference point set
      AxisWarn : Bool := 0;   //   1= Axis warning present
      AxisError : Bool := 0;   //   1= Axis fault present
      Lockout : Bool := 0;   //   1= Axis in lockout state
      ActVelocity : Real := 0.0;   //   Actual drive speed (has to be normed with PNU60000 --> 40000000h = 100%, if BaseSpeedValue is <> 0)
      ActPosition : DInt := 0;   //   Actual position in user unit
      ActMode : Int := 0;   //   Active ModePos mode
      EPosZSW1 : Word := 0;   //   Status of EPOS ZSW1
      EPosZSW2 : Word := 0;   //   Status of EPOS ZSW2
      ActWarn : Word := 0;   //   Actual number of warning
      ActFault : Word := 0;   //   Actual number of error
      Error : Bool := 0;   //   1 = Error present
      Status : Word := 0;   //   Status output (7002 = FB in operation; 8xxx = error description  - read the manual)
      DiagID : Word := 0;   //   Error codes of the cyclic system funtion blocks DPWR / DPRD_DAT
   END_VAR

   VAR 
      stat_Ready4Motion : Bool := 0;   // 1= drive is ready for a new set command
      stat_ExecuteIntern : Bool := 0;   // Internal ExecuteMode signal
      stat_StepHome : UInt;   // step variable for homing
      stat_RetDPRD : Int;   // Static return value for DPRD_DAT
      stat_RetDPWR : Int;   // Static return value for DPWR_DAT
      stat_CycWrite : Struct   // Structure representing the send direction (PLC to drive)
         STW1 : Struct
            jog1 : Bool;   // Bit8
            jog2 : Bool;   // Bit9
            controlByPlc : Bool := TRUE;   // Bit10
            StartHoming : Bool;   // Bit11
            ReleaseBrake : Bool;   // Bit12
            ExternalBlockChange : Bool;   // Bit13
            reserved14 : Bool;   // Bit14
            reserved15 : Bool;   // Bit15
            on : Bool;   // Bit0
            noCoastStop : Bool := TRUE;   // Bit1
            noQuickStop : Bool := TRUE;   // Bit2
            enableOperation : Bool := TRUE;   // Bit3
            cancelTraversing : Bool;   // Bit4
            intermediateStop : Bool;   // Bit5
            activateTraversing : Bool;   // Bit6
            acknowledgeFault : Bool;   // Bit7
         END_STRUCT;
         POS_STW1 : Struct
            MDI_MOD : Bool;   // Bit 8, 1= absolut, 0=relative
            PosModulo : Bool;   // Bit 9, 1=positive direction
            NegModulo : Bool;   // Bit 10, 1=negative direction
            reserved11 : Bool;   // Bit 11
            reserved12 : Bool;   // Bit 12
            reserved13 : Bool;   // Bit 13
            SetupMode : Bool;   // Bit 14, 1=Setup mode activation
            MDI_Activate : Bool;   // Bit 15, 1 =MDI mode activation
            travBlockBit0 : Bool;   // Bit 0
            travBlockBit1 : Bool;   // Bit 1
            travBlockBit2 : Bool;   // Bit 2
            travBlockBit3 : Bool;   // Bit 3
            travBlockBit4 : Bool;   // Bit 4
            travBlockBit5 : Bool;   // Bit 5
            travBlockBit6 : Bool;   // Bit 6
            reserved7 : Bool;   // Bit 7
         END_STRUCT;
         POS_STW2 : Struct
            FlyingRef : Bool;   // Bit 8, 1=Flying referencing activation
            reserved9 : Bool;   // Bit 9,
            SelectProbe : Bool;   // Bit 10, 0=Probe1, 1=Probe2
            ProbeEdgeEval : Bool;   // Bit 11, 0=rising edge, 1=falling edge
            reserved12 : Bool;   // Bit 12
            reserved13 : Bool;   // Bit 13
            "SW-Limit" : Bool;   // Bit 14, 1=Activation of SW-limits
            "HW-Limit" : Bool;   // Bit 15, 1 =Activation of HW-limits
            Trackingmode : Bool;   // Bit 0, 1=Trackingmode
            SetReferencePoint : Bool;   // Bit 1, 1=set reference point
            reserved2 : Bool;   // Bit 2
            reserved3 : Bool;   // Bit 3
            reserved4 : Bool;   // Bit 4
            jog_inc : Bool;   // Bit 5, 1=jog incremental
            reserved6 : Bool;   // Bit 6
            reserved7 : Bool;   // Bit 7
         END_STRUCT;
         STW2 : Struct
            TravelToFixStop : Bool;   // Bit8
            reserved9 : Bool;
            reserved10 : Bool;
            reserved11 : Bool;
            signOfLifeBit0 : Bool;   // Bit12
            signOfLifeBit1 : Bool;   // Bit 13
            signOfLifeBit2 : Bool;   // Bit 14
            signOfLifeBit3 : Bool;   // Bit 15
            reserved0 : Bool;
            reserved1 : Bool;
            reserved2 : Bool;
            reserved3 : Bool;
            reserved4 : Bool;
            reserved5 : Bool;
            reserved6 : Bool;
            reserved7 : Bool;
         END_STRUCT;
         Override : Word;
         MDI_TARPOS : DInt;
         MDI_VELOCITY : DInt;
         MDI_ACC : UInt;
         MDI_DEC : UInt;
         reserved11 : Word;
      END_STRUCT;
      stat_CycRead : Struct   // Structure representing the receiving direction (PLC from drive)
         ZSW1 : Struct
            followingErrorInTolerance : Bool;   // Bit 8
            controlRequest : Bool;   // Bit 9
            targetPosReached : Bool;   // Bit10
            homePosSet : Bool;   // Bit 11
            acknowledgeTraversingBlockActivated : Bool;   // Bit 12
            driveStopped : Bool;   // Bit 13
            axisAccelerates : Bool;   // Bit 14
            axisDecelerates : Bool;   // Bit 15
            readyForSwitchOn : Bool;   // Bit 0
            ready : Bool;   // Bit 1
            operationEnabled : Bool;   // Bit 2
            faultPresent : Bool;   // Bit 3
            noCoastingActive : Bool;   // Bit 4
            noQuickStopActive : Bool;   // Bit 5
            switchingOnInhibitedActive : Bool;   // Bit 6
            warningActive : Bool;   // Bit 7
         END_STRUCT;
         POS_ZSW1 : Word;
         POS_ZSW2 : Word;
         ZSW2 : Struct
            deviceSpecificBit8 : Bool;
            deviceSpecificBit9 : Bool;
            deviceSpecificBit10 : Bool;
            deviceSpecificBit11 : Bool;
            doSignOfLifeBit0 : Bool;
            doSignOfLifeBit1 : Bool;
            doSignOfLifeBit2 : Bool;
            doSignOfLifeBit3 : Bool;
            deviceSpecificBit0 : Bool;
            deviceSpecificBit1 : Bool;
            deviceSpecificBit2 : Bool;
            deviceSpecificBit3 : Bool;
            deviceSpecificBit4 : Bool;
            deviceSpecificBit5 : Bool;
            deviceSpecificBit6 : Bool;
            deviceSpecificBit7 : Bool;
         END_STRUCT;
         MELDW : Word;
         XIST_A : DInt;
         NIST_B : DInt;
         Fault_Code : Word;
         Warn_Code : Word;
         Reserved : Word;
      END_STRUCT;
      stat_ExecAux : Bool;
      stat_ExecR_Trig : Bool;
      stat_Jog1PAux : Bool;
      stat_Jog1PR_trig : Bool;
      stat_Jog2PAux : Bool;
      stat_Jog2PR_trig : Bool;
      stat_Jog1PMode8Aux : Bool;
      stat_Jog1PMode8R_trig : Bool;
      stat_Jog2PMode8Aux : Bool;
      stat_Jog2PMode8R_trig : Bool;
      stat_Status : Word;
      statStartCounter : Int;
      stat_ActMode : Int;
      stat_MaxCounterRetries { ExternalAccessible := 'False'; ExternalVisible := 'False'; ExternalWritable := 'False'} : Int;   // Maximum amount of retries for StartTask
   END_VAR

   VAR_TEMP 
      tempDWord : DWord;   // DWORD for calculation
      tmpSendBuffer : Array[0..11] of Word;   // Buffer to write
      tmpReadBuffer : Array[0..11] of Word;   // Buffer to read
   END_VAR

   VAR CONSTANT 
      MaxCounterStart : Int := 50;   // Maximum cycles for checking ACKStart
      MAXMODE : Int := 8;   // Maximum allowable mode
      STATUS_IN_OPERATION : Word := 16#7002;   // Function block Operational
      ERROR_INVALID_MODE : Word := 16#8202;   // Invalid Mode of Operation selected
      ERROR_OVERRIDE : Word := 16#8203;   // Invalid Override Value
      ERROR_INVALID_TRV_BLOCK : Word := 16#8204;   // Invalid traversing block
      ERROR_DRIVE_ERROR : Word := 16#8401;   // Drive fault
      ERROR_SWITCH_ON_INHIBITED : Word := 16#8402;   // Switch on inhibited
      ERROR_DPRD_DAT : Word := 16#8600;   // Error reading telegram data
      ERROR_DPWR_DAT : Word := 16#8601;   // Error writing telegram data
   END_VAR


BEGIN
	(*############################################################
	    FESTO SE & Co. KG, Esslingen
	    Copyright (c) 2020. All rights reserved.    
	
	    NAME OF FUNCTION BLOCK:         Festo_PTP_Drives_PN
	    VERSION NUMBER:                 V1.5
	    COMPOSER:                       Festo
	    
	    -----------------------------------------------------
	   Date        Name                Activity                                                                              
	   19.03.2020  bkle                created (V1.0)
	   09.03.2021  bkle                name changed
	   18.03.2021  bkle                changed jog behaviour
	   30.07.2021  bkle                Send the StartTask again if ACK is not received - not released
	   06.08.2021  bkle                StartTask is TRUE until ExecuteMode will switch to FALSE
	   22.09.2021  bkle                Added ConfigEpos bits for ReleaseBrake and TravelToFixStop 
	############################################################*)
	
	REGION Check OPM and Override Values
	    // Check the Mode of Operation
	    IF #ModePos > #MAXMODE THEN
	        #Error := True;
	        #stat_Status := #ERROR_INVALID_MODE;
	        #stat_ExecuteIntern := false;
	    ELSIF #ModePos < 1 THEN
	        #Error := True;
	        #stat_Status := #ERROR_INVALID_MODE;
	        #stat_ExecuteIntern := false;
	    ELSE
	        IF #stat_Status = #ERROR_INVALID_MODE THEN
	            #stat_Status := #STATUS_IN_OPERATION;
	            #Error := False;
	        END_IF;
	    END_IF;
	    
	    
	    //Check the Velocity Override 
	    IF (#OverV < 0) OR (#OverV > 199) THEN
	        #stat_Status := #ERROR_OVERRIDE;
	        #Error := True;
	    ELSE
	        // Write Velocity Override into Send Buffer
	        #stat_CycWrite.Override := INT_TO_WORD(REAL_TO_INT(16384.0 * (INT_TO_REAL(#OverV) / 100.0)));
	        IF #stat_Status = #ERROR_OVERRIDE THEN
	            #stat_Status := #STATUS_IN_OPERATION;
	            #Error := False;
	        END_IF;
	    END_IF;
	    
	    //Check the Acceleration Override  (0% - 100%, 100% => W#16#4000)
	    IF (#OverAcc < 0) OR (#OverAcc > 100) THEN
	        #stat_Status := #ERROR_OVERRIDE;
	        #Error := True;
	    ELSE
	        // Write Acceleration Override into Send Buffer
	        #stat_CycWrite.MDI_ACC := INT_TO_WORD(REAL_TO_INT(16384.0 * (INT_TO_REAL(#OverAcc) / 100.0)));
	        IF #stat_Status = #ERROR_OVERRIDE THEN
	            #stat_Status := #STATUS_IN_OPERATION;
	            #Error := False;
	        END_IF;
	    END_IF;
	    
	    //Check the Deceleration Override  (0% - 100%, 100% => W#16#4000)
	    IF (#OverDec < 0) OR (#OverDec > 100) THEN
	        #stat_Status := #ERROR_OVERRIDE;
	        #Error := True;
	    ELSE
	        // Write Deceleration Override into Send Buffer
	        #stat_CycWrite.MDI_DEC := INT_TO_WORD(REAL_TO_INT(16384.0 * (INT_TO_REAL(#OverDec) / 100.0)));
	        IF #stat_Status = #ERROR_OVERRIDE THEN
	            #stat_Status := #STATUS_IN_OPERATION;
	            #Error := False;
	        END_IF;
	    END_IF;
	END_REGION ;
	
	REGION Read Cyclic Data of Telegramm111
	    // Read cyclic telegram 111
	    #stat_RetDPRD := DPRD_DAT(LADDR := #HardwareId,
	                              RECORD => #tmpReadBuffer);
	    
	    //check if the return code is unequal zero -> error occured
	    IF #stat_RetDPRD <> 0 THEN
	        #Error := true;
	        #stat_Status := #ERROR_DPRD_DAT;
	        #DiagID := INT_TO_WORD(#stat_RetDPRD);
	    ELSE
	        
	        // set the Diag status back "in operation"
	        IF #stat_Status = #ERROR_DPRD_DAT THEN
	            #stat_Status := #STATUS_IN_OPERATION;
	            #DiagID := 0;
	            #Error := False;
	        END_IF;
	    END_IF;
	    
	END_REGION ;
	
	
	REGION Read Input from temp data
	    // copy all values from tmp buffer to static data
	    // ZSW1
	    #stat_CycRead.ZSW1.followingErrorInTolerance := #tmpReadBuffer[0].%X8;
	    #stat_CycRead.ZSW1.controlRequest := #tmpReadBuffer[0].%X9;
	    #stat_CycRead.ZSW1.targetPosReached := #tmpReadBuffer[0].%X10;
	    #stat_CycRead.ZSW1.homePosSet := #tmpReadBuffer[0].%X11;
	    #stat_CycRead.ZSW1.acknowledgeTraversingBlockActivated := #tmpReadBuffer[0].%X12;
	    #stat_CycRead.ZSW1.driveStopped := #tmpReadBuffer[0].%X13;
	    #stat_CycRead.ZSW1.axisAccelerates := #tmpReadBuffer[0].%X14;
	    #stat_CycRead.ZSW1.axisDecelerates := #tmpReadBuffer[0].%X15;
	    #stat_CycRead.ZSW1.readyForSwitchOn := #tmpReadBuffer[0].%X0;
	    #stat_CycRead.ZSW1.ready := #tmpReadBuffer[0].%X1;
	    #stat_CycRead.ZSW1.operationEnabled := #tmpReadBuffer[0].%X2;
	    #stat_CycRead.ZSW1.faultPresent := #tmpReadBuffer[0].%X3;
	    #stat_CycRead.ZSW1.noCoastingActive := #tmpReadBuffer[0].%X4;
	    #stat_CycRead.ZSW1.noQuickStopActive := #tmpReadBuffer[0].%X5;
	    #stat_CycRead.ZSW1.switchingOnInhibitedActive := #tmpReadBuffer[0].%X6;
	    #stat_CycRead.ZSW1.warningActive := #tmpReadBuffer[0].%X7;
	    
	    //POS_ZSW1
	    #stat_CycRead.POS_ZSW1 := #tmpReadBuffer[1];
	    #EPosZSW1 := #stat_CycRead.POS_ZSW1;
	    
	    //POS_ZSW2
	    #stat_CycRead.POS_ZSW2 := #tmpReadBuffer[2];
	    #EPosZSW2 := #stat_CycRead.POS_ZSW2;
	    
	    // ZSW2
	    #stat_CycRead.ZSW2.deviceSpecificBit8 := #tmpReadBuffer[3].%X8;
	    #stat_CycRead.ZSW2.deviceSpecificBit9 := #tmpReadBuffer[3].%X9;
	    #stat_CycRead.ZSW2.deviceSpecificBit10 := #tmpReadBuffer[3].%X10;
	    #stat_CycRead.ZSW2.deviceSpecificBit11 := #tmpReadBuffer[3].%X11;
	    #stat_CycRead.ZSW2.doSignOfLifeBit0 := #tmpReadBuffer[3].%X12;
	    #stat_CycRead.ZSW2.doSignOfLifeBit1 := #tmpReadBuffer[3].%X13;
	    #stat_CycRead.ZSW2.doSignOfLifeBit2 := #tmpReadBuffer[3].%X14;
	    #stat_CycRead.ZSW2.doSignOfLifeBit3 := #tmpReadBuffer[3].%X15;
	    #stat_CycRead.ZSW2.deviceSpecificBit0 := #tmpReadBuffer[3].%X0;
	    #stat_CycRead.ZSW2.deviceSpecificBit1 := #tmpReadBuffer[3].%X1;
	    #stat_CycRead.ZSW2.deviceSpecificBit2 := #tmpReadBuffer[3].%X2;
	    #stat_CycRead.ZSW2.deviceSpecificBit3 := #tmpReadBuffer[3].%X3;
	    #stat_CycRead.ZSW2.deviceSpecificBit4 := #tmpReadBuffer[3].%X4;
	    #stat_CycRead.ZSW2.deviceSpecificBit5 := #tmpReadBuffer[3].%X5;
	    #stat_CycRead.ZSW2.deviceSpecificBit6 := #tmpReadBuffer[3].%X6;
	    #stat_CycRead.ZSW2.deviceSpecificBit7 := #tmpReadBuffer[3].%X7;
	    
	    //MELDW
	    #stat_CycRead.MELDW := #tmpReadBuffer[4];
	    
	    //XIST_A
	    #stat_CycRead.XIST_A.%W0 := #tmpReadBuffer[6];
	    #stat_CycRead.XIST_A.%W1 := #tmpReadBuffer[5];
	    
	    //NIST_B
	    #stat_CycRead.NIST_B.%W0 := #tmpReadBuffer[8];
	    #stat_CycRead.NIST_B.%W1 := #tmpReadBuffer[7];
	    
	    //Fault_Code
	    #stat_CycRead.Fault_Code := #tmpReadBuffer[9];
	    
	    //Warn_Code
	    #stat_CycRead.Warn_Code := #tmpReadBuffer[10];
	    
	    //Reserved
	    #stat_CycRead.Reserved := #tmpReadBuffer[11];
	END_REGION ;
	
	// Mapping of the FB Outputs
	#AxisEnabled := #stat_CycRead.ZSW1.operationEnabled;
	#AxisError := #stat_CycRead.ZSW1.faultPresent;
	#AxisWarn := #stat_CycRead.ZSW1.warningActive;
	#AxisPosOk := #stat_CycRead.ZSW1.targetPosReached;
	#AxisRef := #stat_CycRead.ZSW1.homePosSet;
	#AxisAckSetpoint := #stat_CycRead.ZSW1.acknowledgeTraversingBlockActivated;
	#ClampTorqueReached := #stat_CycRead.POS_ZSW2.%X13;
	#AxisSpFixed := #stat_CycRead.ZSW1.driveStopped;
	#ActVelocity := #stat_CycRead.NIST_B;
	
	
	//scaling the ActVelocity output
	IF #BaseSpeedValue <> 0 THEN
	    #ActVelocity := #ActVelocity * ((#BaseSpeedValue / 1073741824.0));
	END_IF;
	
	#ActPosition := #stat_CycRead.XIST_A;
	#ActWarn := #stat_CycRead.Warn_Code;
	#ActFault := #stat_CycRead.Fault_Code;
	#Lockout := #stat_CycRead.ZSW1.switchingOnInhibitedActive;
	
	//Check the drive error and Lockout status
	IF #AxisError THEN
	    #stat_Status := #ERROR_DRIVE_ERROR;
	    #Error := True;
	ELSIF #Lockout THEN
	    #stat_Status := #ERROR_SWITCH_ON_INHIBITED;
	    #Error := True;
	ELSE
	    // error is gone -> set status in operational
	    IF (#stat_Status = #ERROR_DRIVE_ERROR) OR #stat_Status = #ERROR_SWITCH_ON_INHIBITED THEN
	        #stat_Status := #STATUS_IN_OPERATION;
	        #Error := False;
	    END_IF;
	END_IF;
	
	//Enable the Axis
	#stat_CycWrite.STW1.on := #EnableAxis;                       //STW1.0
	
	//fix values for STW1 data
	#stat_CycWrite.STW1.cancelTraversing := #CancelTraversing;   //STW1.4
	#stat_CycWrite.STW1.intermediateStop := #IntermediateStop;   //STW1.5
	#stat_CycWrite.STW1.acknowledgeFault := #AckError;           //STW1.7
	#stat_CycWrite.STW1.controlByPlc := TRUE;                    //STW1.10
	#stat_CycWrite.STW1.enableOperation := TRUE;                 //STW1.3
	
	// copy the position set value into the send struct
	IF #ModePos <> 4 OR #ModePos <> 5 OR #ModePos <> 6 OR #ModePos <> 7 OR #ModePos <> 8 THEN
	    #stat_CycWrite.MDI_TARPOS := #Position;
	ELSE
	    #stat_CycWrite.MDI_TARPOS := 0;
	END_IF;
	
	//copy the velocity set value into the send struct
	#stat_CycWrite.MDI_VELOCITY := #Velocity;
	
	//Jog bits
	// Mode 7
	//Generate the Jog1 Edge
	#stat_Jog1PR_trig := #Jog1 AND NOT #stat_Jog1PAux;
	//Reset the Auxiliary flag 
	#stat_Jog1PAux := #Jog1;
	
	//Generate the Jog2 Edge
	#stat_Jog2PR_trig := #Jog2 AND NOT #stat_Jog2PAux;
	//Reset the Auxiliary flag 
	#stat_Jog2PAux := #Jog2;
	
	//Mode 8
	//Generate the Jog1 Edge
	#stat_Jog1PMode8R_trig := #Jog1 AND NOT #stat_Jog1PMode8Aux;
	//Reset the Auxiliary flag 
	#stat_Jog1PMode8Aux := #Jog1;
	
	//Generate the Jog2 Edge
	#stat_Jog2PMode8R_trig := #Jog2 AND NOT #stat_Jog2PMode8Aux;
	//Reset the Auxiliary flag 
	#stat_Jog2PMode8Aux := #Jog2;
	
	IF #ModePos <> 4 THEN
	    //Start homing
	    #stat_CycWrite.STW1.StartHoming := false;
	END_IF;
	
	//Relative - Absolute
	#stat_CycWrite.POS_STW1.MDI_MOD := false;
	
	//Positive - Negative direction
	#stat_CycWrite.POS_STW1.PosModulo := false;
	#stat_CycWrite.POS_STW1.NegModulo := false;
	
	// setup mode 
	#stat_CycWrite.POS_STW1.SetupMode := false;
	
	// MDI Active
	#stat_CycWrite.POS_STW1.MDI_Activate := false;
	
	//Trackingmode
	#stat_CycWrite.POS_STW2.Trackingmode := false;
	
	//Jog increment
	#stat_CycWrite.POS_STW2.jog_inc := false;
	
	//delete all the record bits
	#stat_CycWrite.POS_STW1.travBlockBit0 := false;
	#stat_CycWrite.POS_STW1.travBlockBit1 := false;
	#stat_CycWrite.POS_STW1.travBlockBit2 := false;
	#stat_CycWrite.POS_STW1.travBlockBit3 := false;
	#stat_CycWrite.POS_STW1.travBlockBit4 := false;
	#stat_CycWrite.POS_STW1.travBlockBit5 := false;
	#stat_CycWrite.POS_STW1.travBlockBit6 := false;
	
	//Check if the drive is ready for a motion
	IF #stat_CycRead.ZSW1.operationEnabled THEN
	    #stat_Ready4Motion := true;
	ELSE
	    #stat_Ready4Motion := false;
	END_IF;
	
	//Generate the Execute Edge for Mode = 4 and 5
	#stat_ExecR_Trig := #ExecuteMode AND NOT #stat_ExecAux;
	//Reset the Auxiliary flag 
	#stat_ExecAux := #ExecuteMode;
	
	// Set the Execute command according to the ModePos
	IF NOT #ExecuteMode THEN
	    #stat_ExecuteIntern := FALSE;
	    #stat_StepHome := 0;
	ELSIF #ExecuteMode AND #stat_Ready4Motion AND NOT (#ModePos = 4 OR #ModePos = 5 OR #ModePos = 7 OR #ModePos = 8) THEN
	    #stat_ExecuteIntern := TRUE;
	    #stat_ActMode := #ModePos;
	    #stat_StepHome := 0;
	ELSIF #stat_ExecR_Trig AND (#ModePos = 4 OR #ModePos = 5) THEN
	    #stat_ActMode := #ModePos;
	    #stat_StepHome := 0;
	ELSIF #ExecuteMode AND (#stat_ActMode = 7 OR #stat_ActMode = 8) THEN
	    #stat_ExecuteIntern := FALSE;
	    #stat_StepHome := 0;
	ELSIF #ExecuteMode AND #ModePos = 4 THEN
	    
	    CASE #stat_StepHome OF
	            
	        0: // homing is active
	            IF NOT #AxisRef THEN
	                #stat_StepHome := 10;
	            ELSIF #AxisError OR (NOT #AxisSpFixed AND #ModePos = 4) THEN
	                #stat_ExecuteIntern := FALSE;
	            END_IF;
	            
	        10: // wait for homing done
	            IF #AxisRef OR #AxisError OR (NOT #stat_Ready4Motion AND #ModePos = 4) OR #ModePos <> #stat_ActMode OR NOT #ExecuteMode THEN
	                #stat_ExecuteIntern := FALSE;
	                #stat_StepHome := 0;
	            END_IF;
	    END_CASE;
	ELSIF #stat_ExecuteIntern AND #ModePos <> #stat_ActMode THEN
	    #stat_ExecuteIntern := false;
	    #stat_StepHome := 0;
	END_IF;
	
	//Reset the jog bits if the ModePos has changed
	IF (#stat_CycWrite.STW1.jog1 OR #stat_CycWrite.STW1.jog2) AND #ModePos <> #stat_ActMode THEN
	    //Set the jog bits to zero
	    #stat_CycWrite.STW1.jog1 := false;
	    #stat_CycWrite.STW1.jog2 := false;
	END_IF;
	
	// Positionig mode with relative movement (MDI)
	IF #ModePos = 1 THEN
	    
	    // Set the MDI bit
	    #stat_CycWrite.POS_STW1.MDI_Activate := true;
	    
	    // positive direction
	    #stat_CycWrite.POS_STW1.PosModulo := #Positive;
	    
	    // #negative direction
	    #stat_CycWrite.POS_STW1.NegModulo := #Negative;
	    
	    // Check if the drive is enabled for a new motion command
	    IF #stat_Ready4Motion THEN
	        
	        IF NOT #stat_CycWrite.STW1.activateTraversing THEN
	            #stat_ExecuteIntern := #stat_ExecR_Trig;
	        END_IF;
	        
	        //Start Traversing Task
	        #stat_CycWrite.STW1.activateTraversing := #stat_ExecuteIntern;
	        
	    END_IF;
	    
	    // Positionig mode with absolute movement (MDI)
	ELSIF #ModePos = 2 THEN
	    
	    // Set the MDI bit
	    #stat_CycWrite.POS_STW1.MDI_Activate := true;
	    
	    //set the Absolute bit
	    #stat_CycWrite.POS_STW1.MDI_MOD := true;
	    
	    // positive direction
	    #stat_CycWrite.POS_STW1.PosModulo := #Positive;
	    
	    // #negative direction
	    #stat_CycWrite.POS_STW1.NegModulo := #Negative;
	    
	    // Check if the drive is enabled for a new motion command
	    IF #stat_Ready4Motion THEN
	        
	        IF NOT #stat_CycWrite.STW1.activateTraversing THEN
	            #stat_ExecuteIntern := #stat_ExecR_Trig;
	        END_IF;
	        
	        //Start Traversing Task
	        #stat_CycWrite.STW1.activateTraversing := #stat_ExecuteIntern;
	        
	    END_IF;
	    
	    // Positioning with setup mode for endless motion
	ELSIF #ModePos = 3 THEN
	    // Set the MDI bit
	    #stat_CycWrite.POS_STW1.MDI_Activate := true;
	    
	    //set the Absolute bit
	    #stat_CycWrite.POS_STW1.MDI_MOD := true;
	    
	    //setup mode
	    #stat_CycWrite.POS_STW1.SetupMode := true;
	    
	    // positive direction
	    #stat_CycWrite.POS_STW1.PosModulo := #Positive;
	    
	    // #negative direction
	    #stat_CycWrite.POS_STW1.NegModulo := #Negative;
	    
	    // Check if the drive is enabled for a new motion command
	    IF #stat_Ready4Motion THEN
	        
	        IF NOT #stat_CycWrite.STW1.activateTraversing THEN
	            #stat_ExecuteIntern := #stat_ExecR_Trig;
	        END_IF;
	        
	        //Start Traversing Task
	        #stat_CycWrite.STW1.activateTraversing := #stat_ExecuteIntern;
	        
	    END_IF;
	    
	    //Homing mode done by the drive due to the parametrized homing method
	ELSIF #ModePos = 4 THEN
	    // positive direction
	    #stat_CycWrite.POS_STW1.PosModulo := #Positive;
	    
	    // #negative direction
	    #stat_CycWrite.POS_STW1.NegModulo := #Negative;
	    
	    // Check if the drive is enabled for a new motion command
	    IF #stat_Ready4Motion THEN
	        
	        //Start homing
	        IF NOT #stat_CycWrite.STW1.StartHoming THEN
	            #stat_ExecuteIntern := #stat_ExecR_Trig;
	        END_IF;
	        
	        #stat_CycWrite.STW1.StartHoming := #stat_ExecuteIntern;
	    END_IF;
	    
	    //set the reference point (actual position)
	ELSIF #ModePos = 5 THEN
	    
	    // check if there is no error in the drive - this function works also when drive is not enabled
	    IF NOT #AxisError THEN
	        
	        //Start homing
	        IF NOT #stat_CycWrite.POS_STW2.SetReferencePoint THEN
	            #stat_ExecuteIntern := #stat_ExecR_Trig;
	        END_IF;
	        //Set the axis zero point
	        #stat_CycWrite.POS_STW2.SetReferencePoint := #stat_ExecuteIntern;
	        
	    END_IF;
	    
	    //Record mode - parametrized records in the drive can be used
	ELSIF #ModePos = 6 THEN
	    
	    //set the position number into the record bits 
	    IF (DINT_TO_INT(#Position) < 0) OR (DINT_TO_INT(#Position) > 127) THEN
	        // Error, wrong record number
	        #stat_Status := #ERROR_INVALID_TRV_BLOCK;
	        #Error := True;
	    ELSE
	        // error is gone -> set status in operational
	        IF #stat_Status = #ERROR_INVALID_TRV_BLOCK THEN
	            #stat_Status := #STATUS_IN_OPERATION;
	            #Error := False;
	        END_IF;
	        
	        // Record bit 0
	        IF (DINT_TO_WORD(#Position) AND W#16#01) = W#16#01 THEN
	            #stat_CycWrite.POS_STW1.travBlockBit0 := true;
	        END_IF;
	        
	        // Record bit 1
	        IF (DINT_TO_WORD(#Position) AND W#16#02) = W#16#02 THEN
	            #stat_CycWrite.POS_STW1.travBlockBit1 := true;
	        END_IF;
	        
	        // Record bit 2
	        IF (DINT_TO_WORD(#Position) AND W#16#04) = W#16#04 THEN
	            #stat_CycWrite.POS_STW1.travBlockBit2 := true;
	        END_IF;
	        
	        // Record bit 3
	        IF (DINT_TO_WORD(#Position) AND W#16#08) = W#16#08 THEN
	            #stat_CycWrite.POS_STW1.travBlockBit3 := true;
	        END_IF;
	        
	        // Record bit 4
	        IF (DINT_TO_WORD(#Position) AND W#16#10) = W#16#10 THEN
	            #stat_CycWrite.POS_STW1.travBlockBit4 := true;
	        END_IF;
	        
	        // Record bit 5
	        IF (DINT_TO_WORD(#Position) AND W#16#20) = W#16#20 THEN
	            #stat_CycWrite.POS_STW1.travBlockBit5 := true;
	        END_IF;
	        
	        // Record bit 6
	        IF (DINT_TO_WORD(#Position) AND W#16#40) = W#16#40 THEN
	            #stat_CycWrite.POS_STW1.travBlockBit6 := true;
	        END_IF;
	        
	        // Check if the drive is enabled for a new motion command
	        IF #stat_Ready4Motion THEN
	            
	            IF NOT #stat_CycWrite.STW1.activateTraversing THEN
	                #stat_ExecuteIntern := #stat_ExecR_Trig;
	            END_IF;
	            
	            //Start Traversing Task
	            #stat_CycWrite.STW1.activateTraversing := #stat_ExecuteIntern;
	            
	        END_IF;
	    END_IF;
	    
	    //Jog mode - positive or negative
	ELSIF #ModePos = 7 THEN
	    
	    // Check if the drive is enabled for a new motion command
	    IF #stat_Ready4Motion THEN
	        
	        IF #stat_Jog1PR_trig AND NOT #Jog2 THEN
	            #stat_CycWrite.STW1.jog1 := TRUE;
	            #stat_ActMode := #ModePos;
	        ELSIF NOT #Jog1 THEN
	            #stat_CycWrite.STW1.jog1 := false;
	        END_IF;
	        
	        IF #stat_Jog2PR_trig AND NOT #Jog1 THEN
	            #stat_CycWrite.STW1.jog2 := TRUE;
	            #stat_ActMode := #ModePos;
	        ELSIF NOT #Jog2 THEN
	            #stat_CycWrite.STW1.jog2 := false;
	        END_IF;
	    ELSE
	        #stat_CycWrite.STW1.jog1 := false;
	        #stat_CycWrite.STW1.jog2 := false;
	        
	    END_IF;
	    
	    // jog incremental mode
	ELSIF #ModePos = 8 THEN
	    
	    // Check if the drive is enabled for a new motion command
	    IF #stat_Ready4Motion THEN
	        
	        //Jog increment
	        #stat_CycWrite.POS_STW2.jog_inc := true;
	        
	        IF #stat_Jog1PMode8R_trig THEN
	            #stat_CycWrite.STW1.jog1 := TRUE;
	            #stat_ActMode := #ModePos;
	        ELSIF NOT #Jog1 THEN
	            #stat_CycWrite.STW1.jog1 := false;
	        END_IF;
	        
	        IF #stat_Jog2PMode8R_trig THEN
	            #stat_CycWrite.STW1.jog2 := TRUE;
	            #stat_ActMode := #ModePos;
	        ELSIF NOT #Jog2 THEN
	            #stat_CycWrite.STW1.jog2 := false;
	        END_IF;
	        
	        IF #stat_Jog1PMode8R_trig AND #stat_Jog2PMode8R_trig THEN
	            #stat_CycWrite.STW1.jog1 := false;
	            #stat_CycWrite.STW1.jog2 := FALSE;
	        END_IF;
	        
	    ELSE
	        #stat_CycWrite.STW1.jog1 := false;
	        #stat_CycWrite.STW1.jog2 := false;
	        
	    END_IF;
	ELSE
	    // modepos < 1 or > 8
	    #stat_ExecuteIntern := false;
	    #stat_CycWrite.STW1.activateTraversing := false;
	    #stat_CycWrite.STW1.StartHoming := false;
	    #stat_CycWrite.POS_STW2.SetReferencePoint := false;
	    #stat_StepHome := 0;
	    #statStartCounter := 0;
	END_IF;
	
	
	REGION ConfigEPos
	    //Maping of the ConfigEPos to the Telegram
	    #stat_CycWrite.STW1.noCoastStop := #ConfigEPos.%X0;         //STW1.1
	    #stat_CycWrite.STW1.noQuickStop := #ConfigEPos.%X1;         //STW1.2
	    #stat_CycWrite.POS_STW2."SW-Limit" := #ConfigEPos.%X2;
	    #stat_CycWrite.POS_STW2."HW-Limit" := #ConfigEPos.%X3;
	    #stat_CycWrite.POS_STW2.ProbeEdgeEval := #ConfigEPos.%X4;
	    #stat_CycWrite.POS_STW2.SelectProbe := #ConfigEPos.%X5;
	    #stat_CycWrite.STW1.ExternalBlockChange := #ConfigEPos.%X6;
	    #stat_CycWrite.POS_STW2.reserved2 := #ConfigEPos.%X7;
	    #stat_CycWrite.POS_STW1.reserved12 := #ConfigEPos.%X8;
	    #stat_CycWrite.STW2.reserved0 := #ConfigEPos.%X9;
	    #stat_CycWrite.STW2.reserved1 := #ConfigEPos.%X10;
	    #stat_CycWrite.STW2.reserved2 := #ConfigEPos.%X11;
	    #stat_CycWrite.STW2.reserved3 := #ConfigEPos.%X12;
	    #stat_CycWrite.STW2.reserved4 := #ConfigEPos.%X13;
	    #stat_CycWrite.STW2.reserved7 := #ConfigEPos.%X14;
	    #stat_CycWrite.STW1.ReleaseBrake := #ReleaseBrake OR #ConfigEPos.%X15;           //STW1.12
	    #stat_CycWrite.STW1.reserved14 := #ConfigEPos.%X16;
	    #stat_CycWrite.STW1.reserved15 := #ConfigEPos.%X17;
	    #stat_CycWrite.POS_STW2.Trackingmode := #ConfigEPos.%X18;    // different mapping to SINA_POS
	    #stat_CycWrite.POS_STW1.reserved7 := #ConfigEPos.%X19;                // reserved
	    #stat_CycWrite.POS_STW1.reserved11 := #ConfigEPos.%X20;               // reserved
	    #stat_CycWrite.POS_STW1.reserved13 := #ConfigEPos.%X21;               // reserved
	    #stat_CycWrite.POS_STW2.reserved13 := #ConfigEPos.%X22;
	    #stat_CycWrite.POS_STW2.reserved4 := #ConfigEPos.%X23;
	    #stat_CycWrite.POS_STW2.reserved6 := #ConfigEPos.%X24;
	    #stat_CycWrite.POS_STW2.reserved7 := #ConfigEPos.%X25;
	    #stat_CycWrite.POS_STW2.reserved12 := #ConfigEPos.%X26;
	    #stat_CycWrite.POS_STW2.reserved13 := #ConfigEPos.%X27;
	    #stat_CycWrite.STW2.reserved5 := #ConfigEPos.%X28;
	    #stat_CycWrite.STW2.reserved6 := #ConfigEPos.%X29;
	    #stat_CycWrite.STW2.TravelToFixStop := #TravelToFixStop OR #ConfigEPos.%X30;     //STW2.8
	    #stat_CycWrite.STW2.reserved9 := #ConfigEPos.%X31;
	END_REGION ;
	
	REGION Write Output to temp data
	    // copy all cyclic data from stat data to tmp buffer
	    ////STW1
	    #tmpSendBuffer[0].%X0 := #stat_CycWrite.STW1.on;
	    #tmpSendBuffer[0].%X1 := #stat_CycWrite.STW1.noCoastStop;
	    #tmpSendBuffer[0].%X2 := #stat_CycWrite.STW1.noQuickStop;
	    #tmpSendBuffer[0].%X3 := #stat_CycWrite.STW1.enableOperation;
	    #tmpSendBuffer[0].%X4 := #stat_CycWrite.STW1.cancelTraversing;
	    #tmpSendBuffer[0].%X5 := #stat_CycWrite.STW1.intermediateStop;
	    #tmpSendBuffer[0].%X6 := #stat_CycWrite.STW1.activateTraversing;
	    #tmpSendBuffer[0].%X7 := #stat_CycWrite.STW1.acknowledgeFault;
	    #tmpSendBuffer[0].%X8 := #stat_CycWrite.STW1.jog1;
	    #tmpSendBuffer[0].%X9 := #stat_CycWrite.STW1.jog2;
	    #tmpSendBuffer[0].%X10 := #stat_CycWrite.STW1.controlByPlc;
	    #tmpSendBuffer[0].%X11 := #stat_CycWrite.STW1.StartHoming;
	    #tmpSendBuffer[0].%X12 := #stat_CycWrite.STW1.ReleaseBrake;
	    #tmpSendBuffer[0].%X13 := #stat_CycWrite.STW1.ExternalBlockChange;
	    #tmpSendBuffer[0].%X14 := #stat_CycWrite.STW1.reserved14;
	    #tmpSendBuffer[0].%X15 := #stat_CycWrite.STW1.reserved15;
	    //POS_STW1
	    #tmpSendBuffer[1].%X0 := #stat_CycWrite.POS_STW1.travBlockBit0;
	    #tmpSendBuffer[1].%X1 := #stat_CycWrite.POS_STW1.travBlockBit1;
	    #tmpSendBuffer[1].%X2 := #stat_CycWrite.POS_STW1.travBlockBit2;
	    #tmpSendBuffer[1].%X3 := #stat_CycWrite.POS_STW1.travBlockBit3;
	    #tmpSendBuffer[1].%X4 := #stat_CycWrite.POS_STW1.travBlockBit4;
	    #tmpSendBuffer[1].%X5 := #stat_CycWrite.POS_STW1.travBlockBit5;
	    #tmpSendBuffer[1].%X6 := #stat_CycWrite.POS_STW1.travBlockBit6;
	    #tmpSendBuffer[1].%X7 := #stat_CycWrite.POS_STW1.reserved7;
	    #tmpSendBuffer[1].%X8 := #stat_CycWrite.POS_STW1.MDI_MOD;
	    #tmpSendBuffer[1].%X9 := #stat_CycWrite.POS_STW1.PosModulo;
	    #tmpSendBuffer[1].%X10 := #stat_CycWrite.POS_STW1.NegModulo;
	    #tmpSendBuffer[1].%X11 := #stat_CycWrite.POS_STW1.reserved11;
	    #tmpSendBuffer[1].%X12 := #stat_CycWrite.POS_STW1.reserved12;
	    #tmpSendBuffer[1].%X13 := #stat_CycWrite.POS_STW1.reserved13;
	    #tmpSendBuffer[1].%X14 := #stat_CycWrite.POS_STW1.SetupMode;
	    #tmpSendBuffer[1].%X15 := #stat_CycWrite.POS_STW1.MDI_Activate;
	    //POS_STW2
	    #tmpSendBuffer[2].%X0 := #stat_CycWrite.POS_STW2.Trackingmode;
	    #tmpSendBuffer[2].%X1 := #stat_CycWrite.POS_STW2.SetReferencePoint;
	    #tmpSendBuffer[2].%X2 := #stat_CycWrite.POS_STW2.reserved2;
	    #tmpSendBuffer[2].%X3 := #stat_CycWrite.POS_STW2.reserved3;
	    #tmpSendBuffer[2].%X4 := #stat_CycWrite.POS_STW2.reserved4;
	    #tmpSendBuffer[2].%X5 := #stat_CycWrite.POS_STW2.jog_inc;
	    #tmpSendBuffer[2].%X6 := #stat_CycWrite.POS_STW2.reserved6;
	    #tmpSendBuffer[2].%X7 := #stat_CycWrite.POS_STW2.reserved7;
	    #tmpSendBuffer[2].%X8 := #stat_CycWrite.POS_STW2.FlyingRef;
	    #tmpSendBuffer[2].%X9 := #stat_CycWrite.POS_STW2.reserved9;
	    #tmpSendBuffer[2].%X10 := #stat_CycWrite.POS_STW2.SelectProbe;
	    #tmpSendBuffer[2].%X11 := #stat_CycWrite.POS_STW2.ProbeEdgeEval;
	    #tmpSendBuffer[2].%X12 := #stat_CycWrite.POS_STW2.reserved12;
	    #tmpSendBuffer[2].%X13 := #stat_CycWrite.POS_STW2.reserved13;
	    #tmpSendBuffer[2].%X14 := #stat_CycWrite.POS_STW2."SW-Limit";
	    #tmpSendBuffer[2].%X15 := #stat_CycWrite.POS_STW2."HW-Limit";
	    //STW2
	    #tmpSendBuffer[3].%X0 := #stat_CycWrite.STW2.reserved0;
	    #tmpSendBuffer[3].%X1 := #stat_CycWrite.STW2.reserved1;
	    #tmpSendBuffer[3].%X2 := #stat_CycWrite.STW2.reserved2;
	    #tmpSendBuffer[3].%X3 := #stat_CycWrite.STW2.reserved3;
	    #tmpSendBuffer[3].%X4 := #stat_CycWrite.STW2.reserved4;
	    #tmpSendBuffer[3].%X5 := #stat_CycWrite.STW2.reserved5;
	    #tmpSendBuffer[3].%X6 := #stat_CycWrite.STW2.reserved6;
	    #tmpSendBuffer[3].%X7 := #stat_CycWrite.STW2.reserved7;
	    #tmpSendBuffer[3].%X8 := #stat_CycWrite.STW2.TravelToFixStop;
	    #tmpSendBuffer[3].%X9 := #stat_CycWrite.STW2.reserved9;
	    #tmpSendBuffer[3].%X10 := #stat_CycWrite.STW2.reserved10;
	    #tmpSendBuffer[3].%X11 := #stat_CycWrite.STW2.reserved11;
	    #tmpSendBuffer[3].%X12 := #stat_CycWrite.STW2.signOfLifeBit0;
	    #tmpSendBuffer[3].%X13 := #stat_CycWrite.STW2.signOfLifeBit1;
	    #tmpSendBuffer[3].%X14 := #stat_CycWrite.STW2.signOfLifeBit2;
	    #tmpSendBuffer[3].%X15 := #stat_CycWrite.STW2.signOfLifeBit3;
	    
	    //Override
	    #tmpSendBuffer[4] := #stat_CycWrite.Override;
	    
	    //TargetPos
	    #tempDWord := DINT_TO_DWORD(#stat_CycWrite.MDI_TARPOS);
	    #tmpSendBuffer[5] := #tempDWord.%W1;
	    #tmpSendBuffer[6] := #tempDWord.%W0;
	    
	    //TargetVelocity
	    #tempDWord := DINT_TO_DWORD(#stat_CycWrite.MDI_VELOCITY);
	    #tmpSendBuffer[7] := #tempDWord.%W1;
	    #tmpSendBuffer[8] := #tempDWord.%W0;
	    
	    // ACC, DEC
	    #tmpSendBuffer[9] := #stat_CycWrite.MDI_ACC;
	    #tmpSendBuffer[10] := #stat_CycWrite.MDI_DEC;
	    #tmpSendBuffer[11] := #stat_CycWrite.reserved11;
	END_REGION ;
	
	REGION Write Cyclic Data of Telegramm 111
	    // Write cyclic telegram 111
	    #stat_RetDPWR := DPWR_DAT(LADDR := #HardwareId,
	                              RECORD := #tmpSendBuffer);
	    
	    // write SETIO status to diagId
	    IF #stat_RetDPWR <> 0 THEN
	        #Error := true;
	        #stat_Status := #ERROR_DPWR_DAT;
	        #DiagID := INT_TO_WORD(#stat_RetDPWR);
	    ELSE
	        // set the Diag status back "in operation"
	        IF #stat_Status = #ERROR_DPWR_DAT THEN
	            #stat_Status := #STATUS_IN_OPERATION;
	            #DiagID := 0;
	            #Error := False;
	        END_IF;
	        
	    END_IF;
	    //Set the Status Output
	    #Status := #stat_Status;
	    #ActMode := #stat_ActMode;
	END_REGION
	
END_FUNCTION_BLOCK

FUNCTION_BLOCK "Festo_ClampingTorque"
TITLE = Festo_ClampingTorque
{ S7_Optimized_Access := 'TRUE' }
AUTHOR : 'Festo SE & Co. KG'
FAMILY : Drives
VERSION : 1.0
//Functin block to write the clamping torque of a Festo drive.
//Linear: percentage of the nominal torque
//Rotative: Absolute value of the torque
   VAR_INPUT 
      Execute { CFC_Visible := 'true'; CFC_ForTest := 'true'} : Bool := 0;   // 1= Execute the function block
      LinearRotative : Bool;   // 1= linear axis 0 = rotative axis
      ClampingTorque : Real := 1.0;   // Torque in Nm for rotative drives
      PercentForce : USInt := 100;   // Percentage of the nominal torque for linear drives
      MAP_HardwareId : HW_IO := 0;   // Hardware ID of the ModuleAccessPoint
   END_VAR

   VAR_OUTPUT 
      Done { CFC_Visible := 'true'; CFC_ForTest := 'true'} : Bool := 1;   // 1= FB finished
      Busy { CFC_Visible := 'true'; CFC_ForTest := 'true'} : Bool := 0;   // 1= FB is busy
      Error { CFC_Visible := 'true'; CFC_ForTest := 'true'} : Bool := 0;   // 1= Error occured while process
      ErrorId { CFC_Visible := 'true'; CFC_ForTest := 'true'} : DWord := 0;   // Number of the error, see  manual
      ErrorString : String[50];   // Errorstring for analyzing
      ActClampingTorque : Real;   // Display the actual written clamping torque
   END_VAR

   VAR 
      ValueWriteREAL { ExternalAccessible := 'False'; ExternalVisible := 'False'; ExternalWritable := 'False'} : Real;
      x { ExternalAccessible := 'False'; ExternalVisible := 'False'; ExternalWritable := 'False'} : Real;
      Festo_PNU_RW_Single_Instance : "Festo_PNU_RW_Single";
      iStep { S7_SetPoint := 'True'} : Int;
      iPNU : Int;
      udGearEnumerator : UDInt;
      udGearDenumerator : UDInt;
      xReadWrite : Bool;
      xStartParam : Bool;
      xBusyParam : Bool;
      xDoneParam : Bool;
      xErrorParam : Bool;
      dwErrorIDParam : DWord;
      lValueReadLint : LInt;
      rValueReadReal : Real;
      rNominalTorque : Real;
      rGearFactor : Real;
      rTorqueFactor : Real;
      trExecuteTrigger {InstructionName := 'R_TRIG'; LibVersion := '1.0'; S7_SetPoint := 'False'} : R_TRIG;
   END_VAR


BEGIN
	(*############################################################
	    FESTO SE & Co. KG, Esslingen
	    Copyright (c) 20203. All rights reserved.    
	
	    NAME OF FUNCTION BLOCK:         Festo_ClampingTorque
	    VERSION NUMBER:                 V1.0
	    COMPOSER:                       Festo
	    
	    -----------------------------------------------------
	   Date        Name                Activity                                                                              
	   03.02.2023  bkle                created (V1.0)
	############################################################*)
	
	#trExecuteTrigger(CLK := #Execute);
	
	//Check the Inputs-hardwareId
	IF #MAP_HardwareId = 0 THEN
	    #Error := true;
	    #ErrorId := 16#00000010;    //HardwareID = 0
	    RETURN;
	END_IF;
	
	//Sequence for reading out the nominal torque and gear ratio
	CASE #iStep OF
	        
	    0: //init
	        #xReadWrite := false;
	        #xStartParam := false;
	        #rGearFactor := 0.0;
	        
	        IF #trExecuteTrigger.Q THEN
	            #Busy := true;
	            #iStep := 10;
	        END_IF;
	        
	    10://read the gear ratio enumerator
	        #iPNU := 11329; //resulting gear enumerator
	        #xStartParam := true;
	        
	        //Check the Inputs-Percent
	        IF #PercentForce = 0 AND #LinearRotative THEN
	            #ErrorId := 1;
	            #ErrorString := 'TargetTorque is zero';
	            #iStep := 999;
	        ELSE
	            #iStep := 15;
	        END_IF;
	        
	    15: //wait for the parameter answer
	        IF #xDoneParam AND NOT #xBusyParam THEN
	            #udGearEnumerator := LINT_TO_UDINT(#lValueReadLint);
	            #xStartParam := FALSE;
	            #iStep := 20;
	        ELSIF #xErrorParam THEN
	            #ErrorId := #dwErrorIDParam;
	            #ErrorString := 'Error in Parameter Channel';
	            #iStep := 999;
	        END_IF;
	        
	    20: //read the gear ration denumerator
	        #iPNU := 11330; //resulting gear enumerator
	        #xStartParam := true;
	        
	        IF #xBusyParam THEN
	            #iStep := 25;
	        END_IF;
	        
	    25: //wait for the parameter answer
	        IF #xDoneParam AND NOT #xBusyParam THEN
	            #udGearDenumerator := LINT_TO_UDINT(#lValueReadLint);
	            #xStartParam := FALSE;
	            #iStep := 30;
	        ELSIF #xErrorParam THEN
	            #ErrorId := #dwErrorIDParam;
	            #ErrorString := 'Error in Parameter Channel';
	            #iStep := 999;
	        END_IF;
	        
	    30: //read the nominal torque of the drive
	        #iPNU := 11704; //resulting nominal torque
	        #xStartParam := true;
	        
	        IF #xBusyParam THEN
	            #iStep := 35;
	        END_IF;
	        
	    35: //wait for the parameter answer
	        IF #xDoneParam AND NOT #xBusyParam THEN
	            #rNominalTorque := #rValueReadReal;
	            #xStartParam := FALSE;
	            #iStep := 100;
	        ELSIF #xErrorParam THEN
	            #ErrorId := #dwErrorIDParam;
	            #ErrorString := 'Error in Parameter Channel';
	            #iStep := 999;
	        END_IF;
	        
	    100: //calculation of the gear ratio
	        #rGearFactor := UDINT_TO_REAL(#udGearEnumerator) / UDINT_TO_REAL(#udGearDenumerator);
	        #rTorqueFactor := #rGearFactor * #rNominalTorque;
	        #iStep := 110;
	        
	    110: //Calculation of clamping torque
	        IF #LinearRotative THEN
	            #ValueWriteREAL := #rTorqueFactor * USINT_TO_REAL(#PercentForce) / 100.0;
	            #iStep := 120;
	        ELSE
	            #ValueWriteREAL := #ClampingTorque;
	            #iStep := 120;
	        END_IF;
	        
	    120: //write the clamping torque
	        #xReadWrite := true;
	        #iPNU := 12168;
	        #ActClampingTorque := #ValueWriteREAL;
	        #xStartParam := true;
	        
	        IF #xBusyParam THEN
	            #iStep := 125;
	        END_IF;
	        
	    125: //wait for the parameter answer
	        IF #xDoneParam AND NOT #xBusyParam THEN
	            #xStartParam := FALSE;
	            #iStep := 200;
	        ELSIF #xErrorParam THEN
	            #ErrorId := #dwErrorIDParam;
	            #ErrorString := 'Error in Parameter Channel';
	            #iStep := 999;
	        END_IF;
	        
	    200: //Done
	        #Done := true;
	        #Busy := false;
	        
	    999: // general error 
	        #Error := true;
	        #Busy := false;
	        #Done := false;
	        
	END_CASE;
	
	//Call PNU_FB
	#Festo_PNU_RW_Single_Instance(Enable := #xStartParam,
	                              ReadWrite := #xReadWrite,
	                              ParameterNo := #iPNU,
	                              Subindex := 0,
	                              ValueWriteREAL := #ValueWriteREAL,
	                              ValueWriteLINT := 0,
	                              ValueWriteBOOL := false,
	                              AxisNo := 16#01,
	                              hardwareId := #MAP_HardwareId,
	                              Busy => #xBusyParam,
	                              Done => #xDoneParam,
	                              ValueReadREAL => #rValueReadReal,
	                              ValueReadLINT => #lValueReadLint,
	                              Error => #xErrorParam,
	                              ErrorId => #dwErrorIDParam);
	
	IF NOT #Execute THEN
	    #iStep := 0;
	    #Busy := false;
	    #Done := false;
	    #Error := false;
	    #ErrorId := 0;
	    #ActClampingTorque := 0;
	    #ErrorString := '';
	END_IF;
	
	
END_FUNCTION_BLOCK

FUNCTION_BLOCK "Festo_PNU_RW_Single"
{ S7_Optimized_Access := 'TRUE' }
VERSION : 0.1
   VAR_INPUT 
      Enable { CFC_Visible := 'true'; CFC_ForTest := 'true'} : Bool := 0;   // 1 = Start the request
      ReadWrite { CFC_Visible := 'true'; CFC_ForTest := 'true'} : Bool := 0;   // 1 = Write, 0 = read
      ParameterNo { CFC_Visible := 'true'; CFC_ForTest := 'true'} : Int := 0;   // PNU number
      Subindex { CFC_Visible := 'true'; CFC_ForTest := 'true'} : Int := 0;   //  Index
      ValueWriteREAL { CFC_Visible := 'true'; CFC_ForTest := 'true'} : Real := 0.0;   // Write value type REAL
      ValueWriteLINT : LInt := 0;   // Write value type LINT
      ValueWriteBOOL : Bool;   // Write value type BOOL
      AxisNo { CFC_Visible := 'true'; CFC_ForTest := 'true'} : Byte := 16#01;   // Axis number
      hardwareId : HW_IO := 0;   // Hardware identifier of the ModuleAccessPoint
   END_VAR

   VAR_OUTPUT 
      Busy { CFC_Visible := 'true'; CFC_ForTest := 'true'} : Bool := 0;   //  1 = function block is busy
      Done { CFC_Visible := 'true'; CFC_ForTest := 'true'} : Bool := 1;   //  1 = request is finished
      ValueReadREAL { CFC_Visible := 'true'; CFC_ForTest := 'true'} : Real := 0.0;   // Read value type REAL
      ValueReadLINT : LInt := 0;   // Read value type LINT
      ValueReadBOOL : Bool;   // Read value type BOOL
      Error { CFC_Visible := 'true'; CFC_ForTest := 'true'} : Bool := 0;   //  1 = Error occured
      ErrorId { CFC_Visible := 'true'; CFC_ForTest := 'true'} : DWord := 0;   // Error number (see manual)
   END_VAR

   VAR 
      st_DataType : Byte := 16#00;   // Format of the parameter
      st_ReqRef : USInt := 16#01;   // Request Referenz ID (1...FF)
      st_step : Int;
      R_TRIG_Execute {InstructionName := 'R_TRIG'; LibVersion := '1.0'} : R_TRIG;
      st_RW_Param : Struct   // Read or write a parameter structure
         ReqHeader : Struct   //  Request header
            ReqRef : Byte := 16#00;   //  Request reference
            ReqId : Byte := 16#01;   //  Request ID 0x1=Read
            AxisNo : Byte := 16#00;   //  Axis (DO-ID number 1 - 254)
            NoParam : Byte := 16#00;   //  No. of parameters (1=single access)
         END_STRUCT;
         ParaAdress : Struct   //  Parameter address
            Attribute : Byte := 16#10;   //  Attribute of parameters (0x10=Value, 0x20=Description, 0x30=Text)
            ElemNo : Byte := 16#01;   //  No. of elements (1=single access)
            ParaNo : Int := 0;   //  Number of parameter (Number 1..65535)
            Index : Int := 0;   //  Subindex (Number 1..65535)
         END_STRUCT;
      END_STRUCT;
      st_WR_Param : Struct   // Structure for writing parameter
         ReqHeader : Struct   //  Request header
            ReqRef : Byte := 16#00;   //  Request reference
            ReqId : Byte := 16#00;   //  Request ID 0x2=write
            AxisNo : Byte := 16#00;   //  Axis (DO-ID number 1 - 254)
            ParaNo : Byte := 16#00;   //  No. of parameters (1=single access)
         END_STRUCT;
         Data : Struct
            Attribute : Byte;
            NoElements : Byte;
            PNU : Int;
            Subindex : Int;
            Value : Array[0..9] of Byte;
         END_STRUCT;
      END_STRUCT;
      st_RD_Param : Struct   // Structure for reading parameter
         RespHeader : Struct   //  Response header
            ReqRefMir : Byte := 16#00;   //  Request reference mirrored
            RespId : Byte := 16#00;   //  Response ID
            AxisNo : Byte := 16#00;   //  Axis (DO-ID number 1 - 254) mirrored
            ParaNo : Byte := 16#00;   //  No. of parameters (1=single access)
         END_STRUCT;
         Data : Struct
            Format : Byte;
            NoValues : Byte;
            Values : Array[0..7] of Byte;
         END_STRUCT;
      END_STRUCT;
      WRREC_Profidrive {InstructionName := 'WRREC'; LibVersion := '1.1'} : WRREC;
      RDREC_Profidrive {InstructionName := 'RDREC'; LibVersion := '1.0'; S7_SetPoint := 'False'} : RDREC;
      st_lenght { S7_SetPoint := 'True'} : UInt;
      st_StatusWR : DWord;   // FB status or error information
      st_StatusRW : DWord;   // FB status or error information
      st_StatusRead : DWord;   // FB status or error information
      st_LenghtRead : UInt;   // Lenght of the data telegramm
   END_VAR
   VAR DB_SPECIFIC
      st_Real_aux : Real;
      st_myRealAT { ExternalAccessible := 'False'; ExternalVisible := 'False'; ExternalWritable := 'False'} AT st_Real_aux : Array[0..3] of Byte;
   END_VAR
   VAR 
      st_ErrorCounter : UInt;
      st_wordhlp : Word;
      IEC_Timer {InstructionName := 'TON_TIME'; LibVersion := '1.0'} : TON_TIME;
      st_StartTimer { S7_SetPoint := 'True'} : Bool;
      st_StartRW : Bool := TRUE;
   END_VAR

   VAR_TEMP 
      tmpWord : Word;   // Temp Word for calculation
      tmpDWord : DWord;   // Temp DWord for calculation
      tmpSINT : SInt;   // Temp SINT for calculation
      tmpINT : Int;   // Temp Int for calculation
      tmpDINT : DInt;   // Temp DINT for calculation
      tmpLINT : LInt;   // Temp LINT for calculation
      i : Int;   // Index variable
   END_VAR

   VAR CONSTANT 
      LenHeader : UInt := 4;   // Lenght of the Header
      LenRequest : UInt := 6;   // Lenght of the Requst telegramm
      LenWrite : UInt := 16;   // Lenght of the Write telegramm
      LenRead : UInt := 10;   // Lenght of the Read telegramm
      PD_Error : DWord := 16#4000_0000;
      MaxRetryCounter : UInt := 150;
   END_VAR


BEGIN
	(*############################################################
	    FESTO SE & Co. KG, Esslingen
	    Copyright (c) 2020. All rights reserved.    
	
	    NAME OF FUNCTION BLOCK:         Festo_PNU_RW_Single
	    VERSION NUMBER:                 V1.0
	    COMPOSER:                       Festo
	    
	    -----------------------------------------------------
	   Date        Name                Activity                                                                              
	   16.02.2021  bkle                created (V1.0)
	############################################################*)
	#R_TRIG_Execute(CLK := #Enable);
	
	//Check the Inputs
	IF #hardwareId = 0 THEN
	    #Error := true;
	    #ErrorId := 16#00001010;    //HardwareID = 0
	    RETURN;
	END_IF;
	
	//Timer
	#IEC_Timer(IN := #st_StartTimer,
	           PT := t#100ms);
	IF #IEC_Timer.Q THEN
	    #st_StartRW := true;
	    #st_StartTimer := false;
	END_IF;
	
	
	CASE #st_step OF
	        
	    0: //Wait for start trigger
	        IF #R_TRIG_Execute.Q THEN
	            #st_StartRW := TRUE;
	            #st_step := 10;
	            #Busy := true;
	        END_IF;
	        
	    10:
	        (* ------------------ HEADER --------------------*)
	        //Fill the Axis number
	        #st_RW_Param.ReqHeader.AxisNo := #AxisNo;
	        
	        // Single parameter access
	        #st_RW_Param.ReqHeader.NoParam := 1;
	        
	        // Requst ID = 1 (Request Parameter)
	        #st_RW_Param.ReqHeader.ReqId := 1;
	        
	        //Request reference starts with 1 and will count up 
	        #st_RW_Param.ReqHeader.ReqRef := #st_ReqRef;
	        
	        (* ------------------ Parameter address ------------*)
	        //Attribute
	        #st_RW_Param.ParaAdress.Attribute := 16#10;
	        
	        //ElemNo.
	        #st_RW_Param.ParaAdress.ElemNo := 1;
	        
	        // Assign PNU
	        #st_RW_Param.ParaAdress.ParaNo := #ParameterNo;
	        
	        // Assign Subindex
	        #st_RW_Param.ParaAdress.Index := #Subindex;
	        
	        // Lenght of the telegramm to be send
	        #st_lenght := #LenHeader + #LenRequest;
	        
	        #WRREC_Profidrive(REQ := #st_StartRW,
	                          ID := #hardwareId,
	                          INDEX := 16#b02e,
	                          LEN := #st_lenght,
	                          STATUS => #st_StatusRW,
	                          RECORD := #st_RW_Param);
	        
	        IF #WRREC_Profidrive.DONE THEN
	            #st_ErrorCounter := 0;
	            //delete old response values
	            #st_RD_Param.RespHeader.ReqRefMir := 0;
	            #st_RD_Param.RespHeader.RespId := 0;
	            #st_RD_Param.RespHeader.AxisNo := 0;
	            #st_RD_Param.RespHeader.ParaNo := 0;
	            #st_RD_Param.Data.Format := 0;
	            #st_RD_Param.Data.NoValues := 0;
	            FOR #i := 0 TO 7 DO
	                #st_RD_Param.Data.Values[#i] := 0;
	            END_FOR;
	            
	            IF NOT #ReadWrite THEN
	                //Read parameter
	                #st_step := 20;
	            ELSE
	                //Write parameter
	                #st_step := 50;
	            END_IF;
	        ELSIF #WRREC_Profidrive.ERROR THEN
	            #tmpWord := DWORD_TO_WORD(SHR(IN := #st_StatusRW, N := 8));
	            #st_wordhlp := #tmpWord;
	            //try it again
	            IF ((#tmpWord = 16#80A7) OR (#tmpWord = 16#80B5) OR (#tmpWord = 16#80C0) OR (#tmpWord = 16#80C1) OR (#tmpWord = 16#80C2)
	                OR (#tmpWord = 16#80C3) OR (#tmpWord = 16#80C4)) AND (#st_ErrorCounter < #MaxRetryCounter) THEN
	                #st_ErrorCounter := #st_ErrorCounter + 1;
	                #st_StartRW := false;
	                #st_StartTimer := TRUE;
	            ELSE
	                #st_step := 70;
	            END_IF;
	            
	        END_IF;
	        
	    20:  //Read Parameter
	        // Lenght of the telegramm for reading
	        #st_lenght := #LenHeader + #LenRead;
	        
	        #RDREC_Profidrive(REQ := #st_StartRW,
	                          ID := #hardwareId,
	                          INDEX := 16#b02e,
	                          MLEN := #st_lenght,
	                          STATUS => #st_StatusRead,
	                          LEN => #st_LenghtRead,
	                          RECORD := #st_RD_Param);
	        
	        IF #RDREC_Profidrive.VALID AND NOT #RDREC_Profidrive.BUSY THEN
	            #st_ErrorCounter := 0;
	            #st_step := 30;
	        ELSIF #RDREC_Profidrive.ERROR THEN
	            #tmpWord := DWORD_TO_WORD(SHR(IN := #st_StatusRead, N := 8));
	            #st_wordhlp := #tmpWord;
	            //try it again
	            IF ((#tmpWord = 16#80A7) OR (#tmpWord = 16#80B5) OR (#tmpWord = 16#80C0) OR (#tmpWord = 16#80C1) OR (#tmpWord = 16#80C2)
	                OR (#tmpWord = 16#80C3) OR (#tmpWord = 16#80C4)) AND (#st_ErrorCounter < #MaxRetryCounter) THEN
	                #st_ErrorCounter := #st_ErrorCounter + 1;
	                #st_StartRW := false;
	                #st_StartTimer := TRUE;
	            ELSE
	                #st_step := 80;
	            END_IF;
	            
	        END_IF;
	        
	    30:  //Reading finished successfull
	        
	        CASE BYTE_TO_INT(#st_RD_Param.Data.Format) OF
	            0:  //reserved
	                #ValueReadREAL := 0;
	                #ValueReadLINT := 0;
	                #ValueReadBOOL := FALSE;
	                
	                #ErrorId := 16#1001;    //reserved DataType
	                // #Error
	                #st_step := 200;
	                
	            1:  // BOOLEAN 
	                //copy the value to the output
	                #ValueReadREAL := 0;
	                #ValueReadLINT := 0;
	                #ValueReadBOOL := BYTE_TO_BOOL(#st_RD_Param.Data.Values[0]);
	                
	                // no error
	                #st_step := 100;
	                
	            2:  //SINT8
	                #tmpSINT := BYTE_TO_SINT(#st_RD_Param.Data.Values[0]);
	                //copy the value to the output
	                #ValueReadREAL := 0;
	                #ValueReadLINT := (SINT_TO_LINT(#tmpSINT));
	                #ValueReadBOOL := FALSE;
	                
	                // no error
	                #st_step := 100;
	                
	            3:  //SINT16
	                #tmpINT.%B0 := #st_RD_Param.Data.Values[1];
	                #tmpINT.%B1 := #st_RD_Param.Data.Values[0];
	                
	                //copy the value to the output
	                #ValueReadREAL := 0;
	                #ValueReadLINT := INT_TO_LINT(#tmpINT);
	                #ValueReadBOOL := FALSE;
	                
	                // no #Error
	                #st_step := 100;
	                
	            4:  //SINT32
	                #tmpDINT.%B0 := #st_RD_Param.Data.Values[3];
	                #tmpDINT.%B1 := #st_RD_Param.Data.Values[2];
	                #tmpDINT.%B2 := #st_RD_Param.Data.Values[1];
	                #tmpDINT.%B3 := #st_RD_Param.Data.Values[0];
	                
	                //copy the value to the output
	                #ValueReadREAL := 0;
	                #ValueReadLINT := DINT_TO_LINT(#tmpDINT);
	                #ValueReadBOOL := FALSE;
	                
	                // no #Error
	                #st_step := 100;
	                
	            5, 65: //USINT8(5) or BYTE(65)
	                //copy the value to the output
	                #ValueReadREAL := 0;
	                #ValueReadLINT := (BYTE_TO_LINT(#st_RD_Param.Data.Values[0]));
	                #ValueReadBOOL := FALSE;
	                
	                // no error
	                #st_step := 100;
	                
	            6, 66: //UINT16(6) or WORD(66)
	                #tmpWord.%B0 := #st_RD_Param.Data.Values[1];
	                #tmpWord.%B1 := #st_RD_Param.Data.Values[0];
	                
	                //copy the value to the output
	                #ValueReadREAL := 0;
	                #ValueReadLINT := WORD_TO_LINT(#tmpWord);
	                #ValueReadBOOL := FALSE;
	                
	                // no #Error
	                #st_step := 100;
	                
	            7, 67: //UDINT32(7) or DWORD(67)
	                #tmpDWord.%B0 := #st_RD_Param.Data.Values[3];
	                #tmpDWord.%B1 := #st_RD_Param.Data.Values[2];
	                #tmpDWord.%B2 := #st_RD_Param.Data.Values[1];
	                #tmpDWord.%B3 := #st_RD_Param.Data.Values[0];
	                
	                //copy the value to the output
	                #ValueReadREAL := 0;
	                #ValueReadLINT := DWORD_TO_LINT(#tmpDWord);
	                #ValueReadBOOL := FALSE;
	                
	                // no #Error
	                #st_step := 100;
	                
	            8:  //FLOAT32
	                #tmpDWord.%B0 := #st_RD_Param.Data.Values[3];
	                #tmpDWord.%B1 := #st_RD_Param.Data.Values[2];
	                #tmpDWord.%B2 := #st_RD_Param.Data.Values[1];
	                #tmpDWord.%B3 := #st_RD_Param.Data.Values[0];
	                
	                //copy the value to the output
	                #ValueReadREAL := DWORD_TO_REAL(#tmpDWord);
	                #ValueReadLINT := 0;
	                #ValueReadBOOL := FALSE;
	                
	                // no #Error
	                #st_step := 100;
	                
	            10:  //OctetString
	                #tmpINT.%B0 := #st_RD_Param.Data.Values[0];
	                #tmpINT.%B1 := #st_RD_Param.Data.Values[1];
	                
	                //copy the value to the output
	                #ValueReadREAL := 0;
	                #ValueReadLINT := INT_TO_LINT(#tmpINT);
	                #ValueReadBOOL := FALSE;
	                
	                // no #Error
	                #st_step := 100;
	                
	                
	            55, 56:  //LINT, ULINT
	                #tmpLINT.%B0 := #st_RD_Param.Data.Values[7];
	                #tmpLINT.%B1 := #st_RD_Param.Data.Values[6];
	                #tmpLINT.%B2 := #st_RD_Param.Data.Values[5];
	                #tmpLINT.%B3 := #st_RD_Param.Data.Values[4];
	                #tmpLINT.%B4 := #st_RD_Param.Data.Values[3];
	                #tmpLINT.%B5 := #st_RD_Param.Data.Values[2];
	                #tmpLINT.%B6 := #st_RD_Param.Data.Values[1];
	                #tmpLINT.%B7 := #st_RD_Param.Data.Values[0];
	                
	                //copy the value to the output
	                #ValueReadREAL := 0;
	                #ValueReadLINT := #tmpLINT;
	                #ValueReadBOOL := FALSE;
	                
	                // no #Error
	                #st_step := 100;
	                
	            68:  //Error
	                #tmpDWord.%B0 := #st_RD_Param.Data.Values[1];
	                #tmpDWord.%B1 := #st_RD_Param.Data.Values[0];
	                #ErrorId := #tmpDWord OR #PD_Error;
	                
	                //copy the value to the output
	                #ValueReadREAL := 0;
	                #ValueReadLINT := 0;
	                #ValueReadBOOL := FALSE;
	                
	                // #Error
	                #st_step := 200;
	                
	            ELSE
	                #ValueReadREAL := 0;
	                #ValueReadLINT := 0;
	                #ValueReadBOOL := FALSE;
	                
	                #ErrorId := 16#1000;    //unknown DataType
	                // #Error
	                #st_step := 200;
	        END_CASE;
	        
	        
	    50: //Write Parameter (First Read dataset then write dataset)
	        // Lenght of the telegramm for reading
	        #st_lenght := #LenHeader + #LenRead;
	        
	        #RDREC_Profidrive(REQ := #st_StartRW,
	                          ID := #hardwareId,
	                          INDEX := 16#b02e,
	                          MLEN := #st_lenght,
	                          STATUS => #st_StatusRead,
	                          LEN => #st_LenghtRead,
	                          RECORD := #st_RD_Param);
	        
	        IF #RDREC_Profidrive.VALID AND NOT #RDREC_Profidrive.BUSY THEN
	            #st_ErrorCounter := 0;
	            #st_step := 55;
	        ELSIF #RDREC_Profidrive.ERROR THEN
	            #tmpWord := DWORD_TO_WORD(SHR(IN := #st_StatusRead, N := 8));
	            #st_wordhlp := #tmpWord;
	            //try it again
	            IF ((#tmpWord = 16#80A7) OR (#tmpWord = 16#80B5) OR (#tmpWord = 16#80C0) OR (#tmpWord = 16#80C1) OR (#tmpWord = 16#80C2)
	                OR (#tmpWord = 16#80C3) OR (#tmpWord = 16#80C4)) AND (#st_ErrorCounter < #MaxRetryCounter) THEN
	                #st_ErrorCounter := #st_ErrorCounter + 1;
	                #st_StartRW := false;
	                #st_StartTimer := TRUE;
	            ELSE
	                #st_step := 80;
	            END_IF;
	        END_IF;
	        
	    55:  //Reading finished
	        CASE BYTE_TO_INT(#st_RD_Param.Data.Format) OF
	            0:  //reserved
	                #ValueReadREAL := 0;
	                #ValueReadLINT := 0;
	                #ValueReadBOOL := FALSE;
	                
	                #ErrorId := 16#1001;    //reserved DataType
	                // #Error
	                #st_step := 200;
	                
	            1, 2, 3, 4, 5, 6, 7, 8, 55, 56, 65, 66, 67:
	                #st_step := 60;
	                
	            68:  //Error
	                #tmpDWord.%B0 := #st_RD_Param.Data.Values[1];
	                #tmpDWord.%B1 := #st_RD_Param.Data.Values[0];
	                #ErrorId := #tmpDWord OR #PD_Error;
	                
	                //copy the value to the output
	                #ValueReadREAL := 0;
	                #ValueReadLINT := 0;
	                #ValueReadBOOL := FALSE;
	                
	                // #Error
	                #st_step := 200;
	                
	            ELSE
	                #ValueReadREAL := 0;
	                #ValueReadLINT := 0;
	                #ValueReadBOOL := FALSE;
	                
	                #ErrorId := 16#1000;    //unknown DataType
	                // #Error
	                #st_step := 200;
	        END_CASE;
	        
	    60:  //reading Done from Write request
	        (* ------------------ HEADER --------------------*)
	        //Fill the Axis number
	        #st_WR_Param.ReqHeader.AxisNo := #AxisNo;
	        
	        // Single parameter access
	        #st_WR_Param.ReqHeader.ParaNo := 1;
	        
	        // Requst ID = 2 (Change Parameter)
	        #st_WR_Param.ReqHeader.ReqId := 2;
	        
	        //Request reference starts with 1 and will count up 
	        #st_WR_Param.ReqHeader.ReqRef := #st_ReqRef + 1;
	        
	        (* ------------------ DATA --------------------*)
	        // Attribute
	        #st_WR_Param.Data.Attribute := 16#10;
	        
	        // Single Access
	        #st_WR_Param.Data.NoElements := 1;
	        
	        // PNU
	        #st_WR_Param.Data.PNU := #ParameterNo;
	        
	        // Subindex
	        #st_WR_Param.Data.Subindex := #Subindex;
	        
	        //Foramt
	        #st_WR_Param.Data.Value[0] := #st_RD_Param.Data.Format;
	        
	        //No. Values
	        #st_WR_Param.Data.Value[1] := 1;
	        
	        //erase send buffer
	        FOR #i := 2 TO 9 DO
	            #st_WR_Param.Data.Value[#i] := 0;
	        END_FOR;
	        
	        CASE BYTE_TO_INT(#st_RD_Param.Data.Format) OF
	            0:  //reserved
	                #ValueReadREAL := 0;
	                #ValueReadLINT := 0;
	                #ValueReadBOOL := FALSE;
	                
	                #ErrorId := 16#1001;    //reserved DataType
	                // #Error
	                #st_step := 200;
	                
	            1:  //BOOL
	                #st_WR_Param.Data.Value[2] := BOOL_TO_BYTE(#ValueWriteBOOL);
	                
	            2, 5, 65:  //SINT8, USINT8, BYTE
	                #st_WR_Param.Data.Value[2] := LINT_TO_BYTE(#ValueWriteLINT);
	                
	            3, 6, 66:  //SINT16, UINT16, WORD
	                #st_WR_Param.Data.Value[2] := #ValueWriteLINT.%B1;
	                #st_WR_Param.Data.Value[3] := #ValueWriteLINT.%B0;
	                
	            4, 7, 67: //SINT32, UDINT32, DWORD
	                #st_WR_Param.Data.Value[2] := #ValueWriteLINT.%B3;
	                #st_WR_Param.Data.Value[3] := #ValueWriteLINT.%B2;
	                #st_WR_Param.Data.Value[4] := #ValueWriteLINT.%B1;
	                #st_WR_Param.Data.Value[5] := #ValueWriteLINT.%B0;
	                
	            8:  //FLOAT32
	                #st_Real_aux := #ValueWriteREAL;
	                #st_WR_Param.Data.Value[2] := #st_myRealAT[0];
	                #st_WR_Param.Data.Value[3] := #st_myRealAT[1];
	                #st_WR_Param.Data.Value[4] := #st_myRealAT[2];
	                #st_WR_Param.Data.Value[5] := #st_myRealAT[3];
	                
	            55, 56:  //SINT64
	                #st_WR_Param.Data.Value[2] := #ValueWriteLINT.%B7;
	                #st_WR_Param.Data.Value[3] := #ValueWriteLINT.%B6;
	                #st_WR_Param.Data.Value[4] := #ValueWriteLINT.%B5;
	                #st_WR_Param.Data.Value[5] := #ValueWriteLINT.%B4;
	                #st_WR_Param.Data.Value[6] := #ValueWriteLINT.%B3;
	                #st_WR_Param.Data.Value[7] := #ValueWriteLINT.%B2;
	                #st_WR_Param.Data.Value[8] := #ValueWriteLINT.%B1;
	                #st_WR_Param.Data.Value[9] := #ValueWriteLINT.%B0;
	                
	        END_CASE;
	        
	        //goto the next step
	        #st_step := 61;
	        
	    61:  //send the write Request
	        // Lenght of the telegramm to be send
	        #st_lenght := #LenHeader + #LenWrite;
	        
	        #WRREC_Profidrive(REQ := #st_StartRW,
	                          ID := #hardwareId,
	                          INDEX := 16#b02e,
	                          LEN := #st_lenght,
	                          STATUS => #st_StatusWR,
	                          RECORD := #st_WR_Param);
	        
	        IF #WRREC_Profidrive.DONE THEN
	            #st_step := 62;
	        ELSIF #WRREC_Profidrive.ERROR THEN
	            #tmpWord := DWORD_TO_WORD(SHR(IN := #st_StatusWR, N := 8));
	            #st_wordhlp := #tmpWord;
	            //try it again
	            IF ((#tmpWord = 16#80A7) OR (#tmpWord = 16#80B5) OR (#tmpWord = 16#80C0) OR (#tmpWord = 16#80C1) OR (#tmpWord = 16#80C2)
	                OR (#tmpWord = 16#80C3) OR (#tmpWord = 16#80C4)) AND (#st_ErrorCounter < #MaxRetryCounter) THEN
	                #st_ErrorCounter := #st_ErrorCounter + 1;
	                #st_StartRW := false;
	                #st_StartTimer := TRUE;
	            ELSE
	                #st_step := 90;
	            END_IF;
	        END_IF;
	        
	    62:  //Read the answer of the write request
	        
	        //delete old response values
	        #st_RD_Param.RespHeader.ReqRefMir := 0;
	        #st_RD_Param.RespHeader.RespId := 0;
	        #st_RD_Param.RespHeader.AxisNo := 0;
	        #st_RD_Param.RespHeader.ParaNo := 0;
	        #st_RD_Param.Data.Format := 0;
	        #st_RD_Param.Data.NoValues := 0;
	        #st_RD_Param.Data.Values[0] := 0;
	        #st_RD_Param.Data.Values[1] := 0;
	        
	        // Lenght of the telegramm for reading
	        #st_lenght := #LenHeader + #LenRead;
	        
	        #RDREC_Profidrive(REQ := #st_StartRW,
	                          ID := #hardwareId,
	                          INDEX := 16#b02e,
	                          MLEN := #st_lenght,
	                          STATUS => #st_StatusRead,
	                          LEN => #st_LenghtRead,
	                          RECORD := #st_RD_Param);
	        
	        IF #RDREC_Profidrive.VALID AND NOT #RDREC_Profidrive.BUSY THEN
	            #st_ErrorCounter := 0;
	            #st_step := 63;
	        ELSIF #RDREC_Profidrive.ERROR THEN
	            #tmpWord := DWORD_TO_WORD(SHR(IN := #st_StatusRead, N := 8));
	            #st_wordhlp := #tmpWord;
	            //try it again
	            IF ((#tmpWord = 16#80A7) OR (#tmpWord = 16#80B5) OR (#tmpWord = 16#80C0) OR (#tmpWord = 16#80C1) OR (#tmpWord = 16#80C2)
	                OR (#tmpWord = 16#80C3) OR (#tmpWord = 16#80C4)) AND (#st_ErrorCounter < #MaxRetryCounter) THEN
	                #st_ErrorCounter := #st_ErrorCounter + 1;
	                #st_StartRW := false;
	                #st_StartTimer := TRUE;
	            ELSE
	                #st_step := 80;
	            END_IF;
	        END_IF;
	        
	    63:  //Reading finished
	        CASE BYTE_TO_INT(#st_RD_Param.RespHeader.RespId) OF
	                
	            2:  //positive resonse
	                #st_step := 150;
	                
	            128..130:  //negative response
	                IF #st_RD_Param.Data.Format = 68 THEN
	                    #tmpDWord.%B0 := #st_RD_Param.Data.Values[1];
	                    #tmpDWord.%B1 := #st_RD_Param.Data.Values[0];
	                    #ErrorId := #tmpDWord OR #PD_Error;
	                    
	                    // #Error
	                    #st_step := 200;
	                ELSE
	                    #ErrorId := 16#1003; //negative response without error code
	                    #st_step := 300;
	                    
	                END_IF;
	            ELSE  //undefined response ID
	                #ErrorId := 16#1002;
	                #st_step := 300;
	        END_CASE;
	        
	    70: // Error while ReadWrite Access
	        #Done := true;
	        #Busy := false;
	        #Error := TRUE;
	        #ErrorId := #st_StatusRW;
	        
